C05463=1079.750,30.402,438.403,173.921,21.272,153.647
C05464=1079.745,30.152,438.419,173.920,21.270,153.647
C05465=1079.739,29.903,438.433,173.919,21.267,153.646
C05466=1079.733,29.653,438.449,173.917,21.266,153.646
C05467=1079.727,29.404,438.464,173.915,21.263,153.646
C05468=1079.722,29.154,438.479,173.914,21.260,153.646
C05469=1079.716,28.905,438.494,173.913,21.258,153.646
C05470=1079.710,28.655,438.509,173.912,21.256,153.645
C05471=1079.703,28.406,438.525,173.910,21.253,153.645
C05472=1079.698,28.157,438.540,173.908,21.251,153.645
C05473=1079.692,27.907,438.555,173.907,21.249,153.645
C05474=1079.686,27.657,438.571,173.906,21.247,153.644
C05475=1079.681,27.408,438.585,173.904,21.244,153.644
C05476=1079.675,27.158,438.601,173.902,21.242,153.644
C05477=1079.669,26.909,438.615,173.901,21.240,153.644
C05478=1079.663,26.659,438.630,173.899,21.237,153.644
C05479=1079.657,26.409,438.646,173.898,21.235,153.643
C05480=1079.651,26.160,438.660,173.897,21.233,153.643
C05481=1079.646,25.910,438.676,173.895,21.230,153.643
C05482=1079.640,25.662,438.690,173.893,21.228,153.643
C05483=1079.634,25.412,438.705,173.892,21.225,153.642
C05484=1079.629,25.163,438.721,173.891,21.223,153.642
C05485=1079.622,24.913,438.736,173.890,21.221,153.642
C05486=1079.617,24.663,438.751,173.887,21.218,153.642
C05487=1079.611,24.414,438.766,173.886,21.216,153.641
C05488=1079.604,24.164,438.781,173.885,21.214,153.641
C05489=1079.599,23.915,438.796,173.884,21.212,153.641
C05490=1079.593,23.665,438.811,173.882,21.209,153.641
C05491=1079.587,23.416,438.825,173.881,21.207,153.641
C05492=1079.581,23.167,438.841,173.879,21.205,153.640
C05493=1079.576,22.918,438.855,173.878,21.202,153.640
C05494=1079.569,22.668,438.870,173.876,21.200,153.640
C05495=1079.564,22.418,438.886,173.875,21.197,153.640
C05496=1079.558,22.169,438.901,173.873,21.195,153.640
C05497=1079.553,21.918,438.915,173.872,21.193,153.639
C05498=1079.547,21.669,438.930,173.870,21.190,153.639
C05499=1079.540,21.420,438.945,173.869,21.188,153.639
C05500=1079.535,21.171,438.960,173.868,21.186,153.639
C05501=1079.529,20.921,438.975,173.866,21.184,153.638
C05502=1079.523,20.672,438.990,173.864,21.181,153.638
C05503=1079.518,20.422,439.005,173.863,21.179,153.638
C05504=1079.512,20.172,439.019,173.862,21.177,153.638
C05505=1079.506,19.923,439.034,173.861,21.174,153.637
C05506=1079.500,19.674,439.048,173.858,21.172,153.637
C05507=1079.494,19.424,439.064,173.857,21.169,153.637
C05508=1079.488,19.175,439.079,173.856,21.167,153.637
C05509=1079.482,18.925,439.094,173.855,21.165,153.637
C05510=1079.477,18.676,439.107,173.853,21.162,153.636
C05511=1079.470,18.426,439.122,173.851,21.161,153.636
C05512=1079.465,18.177,439.138,173.850,21.158,153.636
C05513=1079.459,17.927,439.152,173.849,21.156,153.636
C05514=1079.453,17.677,439.166,173.847,21.153,153.635
C05515=1079.447,17.428,439.181,173.846,21.151,153.635
C05516=1079.442,17.179,439.196,173.844,21.149,153.635
C05517=1079.436,16.930,439.211,173.843,21.147,153.635
C05518=1079.430,16.679,439.225,173.841,21.144,153.635
C05519=1079.424,16.430,439.240,173.840,21.142,153.634
C05520=1079.418,16.181,439.255,173.839,21.139,153.634
C05521=1079.412,15.932,439.269,173.837,21.137,153.634
C05522=1079.407,15.681,439.284,173.836,21.135,153.634
C05523=1079.401,15.432,439.299,173.834,21.133,153.634
C05524=1079.395,15.154,439.315,173.833,21.130,153.633
C05525=1079.388,14.875,439.332,173.831,21.127,153.633
C05526=1079.382,14.596,439.348,173.830,21.125,153.633
C05527=1079.375,14.317,439.364,173.828,21.122,153.633
C05528=1079.369,14.068,439.378,173.826,21.120,153.632
C05529=1079.362,13.819,439.393,173.825,21.118,153.632
C05530=1079.357,13.569,439.407,173.824,21.116,153.632
C05531=1079.351,13.320,439.422,173.822,21.113,153.632
C05532=1079.345,13.070,439.436,173.820,21.111,153.631
C05533=1079.339,12.820,439.451,173.819,21.108,153.631
C05534=1079.333,12.571,439.465,173.818,21.106,153.631
C05535=1079.327,12.321,439.480,173.816,21.104,153.631
C05536=1079.321,12.072,439.494,173.815,21.102,153.631
C05537=1079.315,11.822,439.508,173.813,21.100,153.630
C05538=1079.309,11.573,439.523,173.812,21.097,153.630
C05539=1079.303,11.324,439.538,173.811,21.095,153.630
C05540=1079.297,11.074,439.552,173.809,21.092,153.630
C05541=1079.292,10.825,439.566,173.808,21.090,153.630
C05542=1079.285,10.574,439.581,173.806,21.088,153.629
C05543=1079.280,10.326,439.595,173.805,21.086,153.629
C05544=1079.274,10.075,439.609,173.803,21.083,153.629
C05545=1079.268,9.826,439.624,173.802,21.081,153.629
C05546=1079.262,9.577,439.638,173.801,21.079,153.628
C05547=1079.256,9.327,439.653,173.799,21.077,153.628
C05548=1079.250,9.077,439.667,173.797,21.074,153.628
C05549=1079.244,8.828,439.682,173.796,21.072,153.628
C05550=1079.239,8.578,439.695,173.795,21.070,153.628
C05551=1079.233,8.329,439.710,173.793,21.068,153.627
C05552=1079.227,8.079,439.724,173.792,21.066,153.627
C05553=1079.221,7.830,439.739,173.790,21.063,153.627
C05554=1079.216,7.580,439.753,173.789,21.061,153.627
C05555=1079.209,7.331,439.768,173.788,21.058,153.626
C05556=1079.204,7.081,439.782,173.786,21.056,153.626
C05557=1079.197,6.833,439.795,173.784,21.053,153.626
C05558=1079.191,6.582,439.810,173.783,21.051,153.626
C05559=1079.186,6.333,439.824,173.782,21.049,153.626
C05560=1079.180,6.084,439.838,173.781,21.047,153.625
C05561=1079.174,5.834,439.852,173.779,21.045,153.625
C05562=1079.168,5.585,439.867,173.777,21.042,153.625
C05563=1079.162,5.335,439.881,173.776,21.040,153.625
C05564=1079.156,5.085,439.895,173.775,21.038,153.625
C05565=1079.151,4.836,439.910,173.774,21.036,153.624
C05566=1079.145,4.586,439.924,173.772,21.034,153.624
C05567=1079.139,4.336,439.938,173.770,21.031,153.624
C05568=1079.133,4.087,439.952,173.769,21.029,153.624
C05569=1079.127,3.838,439.966,173.768,21.026,153.623
C05570=1079.121,3.588,439.981,173.766,21.024,153.623
C05571=1079.115,3.338,439.994,173.764,21.021,153.623
C05572=1079.110,3.089,440.008,173.763,21.019,153.623
C05573=1079.104,2.839,440.022,173.762,21.017,153.623
C05574=1079.098,2.590,440.037,173.761,21.015,153.622
C05575=1079.092,2.340,440.051,173.759,21.013,153.622
C05576=1079.086,2.091,440.064,173.757,21.010,153.622
C05577=1079.080,1.842,440.079,173.756,21.008,153.622
C05578=1079.074,1.592,440.093,173.755,21.005,153.622
C05579=1079.069,1.342,440.107,173.754,21.004,153.621
C05580=1079.063,1.092,440.121,173.752,21.002,153.621
C05581=1079.058,0.843,440.135,173.750,20.999,153.621
C05582=1079.051,0.593,440.150,173.749,20.997,153.621
C05583=1079.045,0.344,440.163,173.748,20.994,153.620
C05584=1079.040,0.094,440.177,173.747,20.992,153.620
C05585=1079.034,-0.155,440.191,173.745,20.989,153.620
C05586=1079.028,-0.405,440.206,173.743,20.987,153.620
C05587=1079.022,-0.654,440.219,173.742,20.985,153.620
C05588=1079.017,-0.931,440.234,173.741,20.983,153.619
C05589=1079.010,-1.208,440.251,173.739,20.980,153.619
C05590=1079.003,-1.484,440.265,173.738,20.977,153.619
C05591=1078.996,-1.761,440.281,173.736,20.975,153.619
C05592=1078.991,-2.011,440.295,173.734,20.972,153.618
C05593=1078.985,-2.260,440.309,173.733,20.970,153.618
C05594=1078.980,-2.510,440.323,173.732,20.968,153.618
C05595=1078.974,-2.759,440.336,173.730,20.966,153.618
C05596=1078.968,-3.009,440.350,173.729,20.963,153.618
C05597=1078.962,-3.258,440.365,173.727,20.961,153.617
C05598=1078.956,-3.508,440.379,173.726,20.959,153.617
C05599=1078.950,-3.757,440.392,173.725,20.957,153.617
C05600=1078.945,-4.007,440.406,173.723,20.954,153.617
C05601=1078.938,-4.257,440.420,173.721,20.952,153.617
C05602=1078.932,-4.506,440.434,173.720,20.950,153.616
C05603=1078.927,-4.756,440.447,173.719,20.948,153.616
C05604=1078.921,-5.005,440.461,173.718,20.946,153.616
C05605=1078.915,-5.255,440.475,173.716,20.943,153.616
C05606=1078.908,-5.505,440.488,173.714,20.941,153.616
C05607=1078.903,-5.754,440.502,173.713,20.939,153.615
C05608=1078.897,-6.004,440.516,173.712,20.937,153.615
C05609=1078.891,-6.252,440.530,173.711,20.934,153.615
C05610=1078.885,-6.503,440.544,173.708,20.932,153.615
C05611=1078.879,-6.752,440.557,173.707,20.930,153.615
C05612=1078.873,-7.002,440.571,173.706,20.928,153.614
C05613=1078.867,-7.251,440.585,173.705,20.926,153.614
C05614=1078.862,-7.500,440.598,173.703,20.924,153.614
C05615=1078.855,-7.750,440.612,173.701,20.921,153.614
C05616=1078.849,-8.000,440.626,173.700,20.919,153.614
C05617=1078.843,-8.249,440.639,173.699,20.917,153.613
C05618=1078.838,-8.499,440.653,173.698,20.914,153.613
C05619=1078.832,-8.749,440.666,173.696,20.912,153.613
C05620=1078.826,-8.998,440.679,173.695,20.910,153.613
C05621=1078.821,-9.248,440.693,173.693,20.907,153.612
C05622=1078.814,-9.497,440.707,173.692,20.905,153.612
C05623=1078.808,-9.747,440.721,173.690,20.903,153.612
C05624=1078.802,-9.997,440.734,173.689,20.901,153.612
C05625=1078.797,-10.246,440.748,173.688,20.899,153.612
C05626=1078.790,-10.495,440.761,173.686,20.896,153.612
C05627=1078.785,-10.745,440.775,173.684,20.895,153.611
C05628=1078.779,-10.994,440.788,173.683,20.892,153.611
C05629=1078.773,-11.244,440.802,173.682,20.890,153.611
C05630=1078.767,-11.493,440.815,173.681,20.888,153.611
C05631=1078.761,-11.744,440.829,173.679,20.885,153.611
C05632=1078.755,-11.993,440.842,173.677,20.883,153.610
C05633=1078.750,-12.243,440.856,173.676,20.881,153.610
C05634=1078.743,-12.492,440.869,173.675,20.879,153.610
C05635=1078.738,-12.742,440.883,173.674,20.877,153.610
C05636=1078.732,-12.991,440.897,173.672,20.874,153.610
C05637=1078.727,-13.241,440.910,173.670,20.872,153.609
C05638=1078.720,-13.490,440.923,173.669,20.870,153.609
C05639=1078.715,-13.740,440.937,173.668,20.868,153.609
C05640=1078.709,-13.989,440.950,173.666,20.866,153.609
C05641=1078.703,-14.239,440.964,173.665,20.863,153.608
C05642=1078.697,-14.488,440.977,173.663,20.861,153.608
C05643=1078.692,-14.738,440.990,173.662,20.859,153.608
C05644=1078.686,-14.988,441.004,173.661,20.856,153.608
C05645=1078.679,-15.238,441.017,173.659,20.854,153.608
C05646=1078.673,-15.487,441.031,173.658,20.852,153.608
C05647=1078.667,-15.737,441.044,173.656,20.850,153.607
C05648=1078.661,-15.986,441.057,173.655,20.848,153.607
C05649=1078.656,-16.236,441.071,173.654,20.846,153.607
C05650=1078.649,-16.485,441.084,173.652,20.844,153.607
C05651=1078.644,-16.735,441.097,173.651,20.842,153.607
C05652=1078.637,-17.010,441.111,173.649,20.839,153.606
C05653=1078.631,-17.285,441.126,173.648,20.837,153.606
C05654=1078.624,-17.560,441.141,173.646,20.835,153.606
C05655=1078.617,-17.835,441.155,173.644,20.832,153.606
C05656=1078.612,-18.085,441.168,173.643,20.830,153.606
C05657=1078.605,-18.334,441.181,173.642,20.828,153.605
C05658=1078.600,-18.584,441.195,173.640,20.826,153.605
C05659=1078.593,-18.834,441.208,173.639,20.823,153.605
C05660=1078.587,-19.083,441.221,173.637,20.821,153.605
C05661=1078.581,-19.333,441.235,173.636,20.819,153.605
C05662=1078.576,-19.583,441.248,173.634,20.817,153.605
C05663=1078.570,-19.832,441.261,173.633,20.815,153.604
C05664=1078.563,-20.081,441.274,173.632,20.812,153.604
C05665=1078.557,-20.331,441.287,173.630,20.810,153.604
C05666=1078.552,-20.581,441.301,173.629,20.808,153.604
C05667=1078.546,-20.830,441.314,173.627,20.806,153.604
C05668=1078.540,-21.080,441.327,173.626,20.804,153.603
C05669=1078.534,-21.329,441.340,173.625,20.802,153.603
C05670=1078.528,-21.579,441.353,173.624,20.800,153.603
C05671=1078.522,-21.829,441.366,173.621,20.797,153.603
C05672=1078.516,-22.079,441.379,173.620,20.795,153.603
C05673=1078.510,-22.328,441.392,173.619,20.793,153.603
C05674=1078.505,-22.577,441.406,173.618,20.791,153.602
C05675=1078.499,-22.827,441.418,173.616,20.789,153.602
C05676=1078.493,-23.076,441.431,173.615,20.787,153.602
C05677=1078.487,-23.326,441.444,173.613,20.784,153.602
C05678=1078.481,-23.575,441.457,173.612,20.782,153.602
C05679=1078.476,-23.825,441.470,173.610,20.780,153.601
C05680=1078.470,-24.074,441.484,173.609,20.778,153.601
C05681=1078.464,-24.324,441.496,173.608,20.776,153.601
C05682=1078.458,-24.574,441.509,173.607,20.774,153.601
C05683=1078.452,-24.823,441.522,173.604,20.772,153.601
C05684=1078.446,-25.073,441.536,173.603,20.770,153.601
C05685=1078.440,-25.323,441.548,173.602,20.767,153.600
C05686=1078.434,-25.572,441.562,173.601,20.765,153.600
C05687=1078.428,-25.822,441.574,173.599,20.763,153.600
C05688=1078.422,-26.072,441.587,173.598,20.761,153.600
C05689=1078.417,-26.322,441.601,173.597,20.759,153.600
C05690=1078.411,-26.571,441.613,173.594,20.757,153.599
C05691=1078.405,-26.820,441.626,173.593,20.754,153.599
C05692=1078.399,-27.070,441.639,173.592,20.752,153.599
C05693=1078.393,-27.319,441.652,173.591,20.750,153.599
C05694=1078.387,-27.569,441.665,173.589,20.748,153.599
C05695=1078.381,-27.819,441.677,173.588,20.746,153.599
C05696=1078.375,-28.068,441.690,173.586,20.744,153.598
C05697=1078.369,-28.318,441.703,173.585,20.742,153.598
C05698=1078.363,-28.567,441.716,173.583,20.740,153.598
C05699=1078.357,-28.817,441.729,173.582,20.738,153.598
C05700=1078.351,-29.067,441.741,173.581,20.736,153.598
C05701=1078.345,-29.316,441.755,173.579,20.734,153.598
C05702=1078.339,-29.566,441.767,173.578,20.732,153.597
C05703=1078.333,-29.816,441.780,173.576,20.730,153.597
C05704=1078.327,-30.065,441.793,173.575,20.728,153.597
C05705=1078.322,-30.315,441.805,173.573,20.726,153.597
C05706=1078.316,-30.564,441.818,173.572,20.723,153.597
C05707=1078.309,-30.814,441.831,173.571,20.721,153.597
C05708=1078.304,-31.064,441.843,173.570,20.719,153.596
C05709=1078.298,-31.313,441.856,173.567,20.717,153.596
C05710=1078.292,-31.563,441.869,173.566,20.715,153.596
C05711=1078.285,-31.813,441.882,173.565,20.713,153.596
C05712=1078.280,-32.063,441.894,173.564,20.711,153.596
C05713=1078.273,-32.312,441.906,173.562,20.709,153.596
C05714=1078.267,-32.561,441.919,173.561,20.707,153.595
C05715=1078.261,-32.811,441.932,173.560,20.705,153.595
C05716=1078.255,-33.085,441.946,173.557,20.702,153.595
C05717=1078.248,-33.359,441.960,173.556,20.700,153.595
C05718=1078.242,-33.634,441.973,173.555,20.698,153.595
C05719=1078.235,-33.908,441.987,173.553,20.695,153.595
C05720=1078.229,-34.158,442.000,173.552,20.693,153.594
C05721=1078.223,-34.407,442.013,173.550,20.691,153.594
C05722=1078.218,-34.656,442.025,173.549,20.690,153.594
C05723=1078.212,-34.906,442.038,173.548,20.688,153.594
C05724=1078.206,-35.156,442.050,173.546,20.686,153.594
C05725=1078.200,-35.406,442.063,173.544,20.683,153.594
C05726=1078.194,-35.655,442.076,173.543,20.681,153.593
C05727=1078.188,-35.905,442.089,173.542,20.679,153.593
C05728=1078.183,-36.154,442.101,173.540,20.677,153.593
C05729=1078.177,-36.404,442.113,173.539,20.675,153.593
C05730=1078.171,-36.654,442.126,173.538,20.673,153.593
C05731=1078.164,-36.904,442.138,173.536,20.671,153.593
C05732=1078.159,-37.153,442.150,173.534,20.669,153.593
C05733=1078.153,-37.403,442.163,173.533,20.667,153.592
C05734=1078.147,-37.652,442.176,173.532,20.665,153.592
C05735=1078.141,-37.902,442.188,173.530,20.663,153.592
C05736=1078.135,-38.152,442.201,173.529,20.661,153.592
C05737=1078.130,-38.401,442.213,173.528,20.659,153.592
C05738=1078.124,-38.651,442.226,173.526,20.657,153.592
C05739=1078.117,-38.900,442.238,173.524,20.654,153.591
C05740=1078.111,-39.150,442.250,173.523,20.652,153.591
C05741=1078.105,-39.400,442.263,173.522,20.650,153.591
C05742=1078.099,-39.649,442.274,173.520,20.649,153.591
C05743=1078.093,-39.899,442.287,173.519,20.647,153.591
C05744=1078.087,-40.149,442.299,173.517,20.645,153.591
C05745=1078.081,-40.399,442.312,173.516,20.643,153.591
C05746=1078.075,-40.647,442.324,173.515,20.641,153.590
C05747=1078.070,-40.897,442.336,173.513,20.639,153.590
C05748=1078.064,-41.147,442.349,173.511,20.637,153.590
C05749=1078.057,-41.397,442.361,173.510,20.635,153.590
C05750=1078.051,-41.647,442.373,173.509,20.633,153.590
C05751=1078.046,-41.896,442.385,173.507,20.631,153.590
C05752=1078.039,-42.145,442.397,173.506,20.629,153.590
C05753=1078.033,-42.395,442.410,173.505,20.627,153.589
C05754=1078.027,-42.645,442.422,173.503,20.625,153.589
C05755=1078.022,-42.894,442.435,173.501,20.623,153.589
C05756=1078.015,-43.144,442.447,173.500,20.621,153.589
C05757=1078.009,-43.394,442.459,173.498,20.619,153.589
C05758=1078.004,-43.644,442.472,173.497,20.617,153.589
C05759=1077.997,-43.893,442.483,173.496,20.615,153.588
C05760=1077.992,-44.142,442.496,173.494,20.614,153.588
C05761=1077.986,-44.392,442.508,173.493,20.612,153.588
C05762=1077.980,-44.641,442.520,173.492,20.610,153.588
C05763=1077.974,-44.891,442.533,173.490,20.608,153.588
C05764=1077.967,-45.141,442.545,173.488,20.605,153.588
C05765=1077.961,-45.391,442.556,173.487,20.603,153.588
C05766=1077.956,-45.640,442.569,173.485,20.602,153.588
C05767=1077.950,-45.890,442.581,173.484,20.600,153.588
C05768=1077.944,-46.140,442.593,173.483,20.598,153.587
C05769=1077.938,-46.389,442.605,173.482,20.596,153.587
C05770=1077.932,-46.639,442.617,173.480,20.594,153.587
C05771=1077.926,-46.888,442.630,173.479,20.592,153.587
C05772=1077.920,-47.138,442.642,173.478,20.590,153.587
C05773=1077.914,-47.388,442.653,173.475,20.588,153.587
C05774=1077.908,-47.638,442.666,173.474,20.586,153.587
C05775=1077.902,-47.887,442.677,173.473,20.584,153.586
C05776=1077.896,-48.136,442.690,173.471,20.582,153.586
C05777=1077.890,-48.386,442.702,173.470,20.580,153.586
C05778=1077.885,-48.636,442.713,173.469,20.578,153.586
C05779=1077.879,-48.886,442.726,173.467,20.576,153.586
C05780=1077.873,-49.160,442.739,173.465,20.574,153.586
C05781=1077.866,-49.435,442.752,173.464,20.572,153.586
C05782=1077.859,-49.709,442.766,173.462,20.570,153.585
C05783=1077.852,-49.984,442.779,173.461,20.568,153.585
C05784=1077.847,-50.234,442.791,173.459,20.566,153.585
C05785=1077.841,-50.483,442.803,173.458,20.564,153.585
C05786=1077.834,-50.733,442.815,173.456,20.562,153.585
C05787=1077.829,-50.982,442.827,173.455,20.560,153.585
C05788=1077.822,-51.232,442.838,173.454,20.558,153.585
C05789=1077.816,-51.482,442.850,173.452,20.557,153.585
C05790=1077.810,-51.732,442.862,173.451,20.555,153.584
C05791=1077.804,-51.981,442.874,173.449,20.553,153.584
C05792=1077.797,-52.231,442.885,173.448,20.551,153.584
C05793=1077.792,-52.481,442.898,173.447,20.549,153.584
C05794=1077.786,-52.730,442.909,173.444,20.547,153.584
C05795=1077.779,-52.980,442.921,173.443,20.545,153.584
C05796=1077.773,-53.230,442.933,173.442,20.543,153.584
C05797=1077.767,-53.479,442.945,173.440,20.542,153.584
C05798=1077.761,-53.729,442.956,173.439,20.540,153.584
C05799=1077.755,-53.979,442.969,173.438,20.538,153.583
C05800=1077.749,-54.227,442.980,173.436,20.537,153.583
C05801=1077.743,-54.478,442.991,173.435,20.535,153.583
C05802=1077.737,-54.728,443.004,173.433,20.533,153.583
C05803=1077.731,-54.977,443.015,173.432,20.531,153.583
C05804=1077.724,-55.227,443.027,173.431,20.529,153.583
C05805=1077.719,-55.476,443.039,173.428,20.527,153.583
C05806=1077.713,-55.726,443.050,173.427,20.525,153.583
C05807=1077.706,-55.976,443.062,173.426,20.523,153.583
C05808=1077.700,-56.225,443.073,173.424,20.522,153.583
C05809=1077.694,-56.475,443.086,173.423,20.520,153.582
C05810=1077.688,-56.724,443.097,173.421,20.518,153.582
C05811=1077.682,-56.974,443.109,173.420,20.516,153.582
C05812=1077.676,-57.224,443.121,173.418,20.515,153.582
C05813=1077.670,-57.473,443.132,173.417,20.513,153.582
C05814=1077.664,-57.723,443.144,173.416,20.511,153.582
C05815=1077.658,-57.972,443.155,173.414,20.510,153.582
C05816=1077.652,-58.222,443.167,173.413,20.508,153.582
C05817=1077.646,-58.473,443.179,173.412,20.506,153.582
C05818=1077.640,-58.721,443.190,173.409,20.504,153.582
C05819=1077.634,-58.972,443.202,173.408,20.502,153.582
C05820=1077.628,-59.221,443.214,173.407,20.500,153.581
C05821=1077.622,-59.471,443.225,173.405,20.498,153.581
C05822=1077.616,-59.720,443.236,173.404,20.497,153.581
C05823=1077.610,-59.970,443.248,173.402,20.495,153.581
C05824=1077.603,-60.220,443.260,173.401,20.493,153.581
C05825=1077.598,-60.469,443.271,173.400,20.491,153.581
C05826=1077.591,-60.719,443.283,173.398,20.490,153.581
C05827=1077.586,-60.969,443.295,173.397,20.488,153.581
C05828=1077.579,-61.218,443.307,173.395,20.486,153.581
C05829=1077.574,-61.468,443.317,173.394,20.484,153.580
C05830=1077.567,-61.718,443.329,173.392,20.483,153.580
C05831=1077.561,-61.967,443.340,173.391,20.481,153.580
C05832=1077.556,-62.217,443.352,173.389,20.479,153.580
C05833=1077.550,-62.466,443.364,173.388,20.477,153.580
C05834=1077.543,-62.716,443.375,173.386,20.475,153.580
C05835=1077.537,-62.966,443.386,173.385,20.474,153.580
C05836=1077.532,-63.216,443.398,173.383,20.472,153.580
C05837=1077.526,-63.465,443.409,173.382,20.470,153.580
C05838=1077.519,-63.715,443.421,173.381,20.468,153.580
C05839=1077.513,-63.964,443.432,173.379,20.467,153.580
C05840=1077.507,-64.215,443.443,173.378,20.465,153.579
C05841=1077.502,-64.464,443.455,173.376,20.463,153.579
C05842=1077.495,-64.714,443.467,173.375,20.461,153.579
C05843=1077.490,-64.963,443.478,173.373,20.460,153.579
C05844=1077.483,-65.239,443.490,173.371,20.457,153.579
C05845=1077.476,-65.515,443.503,173.370,20.456,153.579
C05846=1077.470,-65.791,443.516,173.368,20.454,153.579
C05847=1077.463,-66.067,443.528,173.367,20.452,153.579
C05848=1077.457,-66.317,443.539,173.366,20.451,153.579
C05849=1077.451,-66.566,443.551,173.364,20.449,153.579
C05850=1077.445,-66.816,443.562,173.362,20.447,153.579
C05851=1077.439,-67.066,443.574,173.360,20.445,153.579
C05852=1077.434,-67.316,443.585,173.359,20.443,153.578
C05853=1077.428,-67.564,443.596,173.358,20.442,153.578
C05854=1077.421,-67.815,443.608,173.356,20.440,153.578
C05855=1077.416,-68.064,443.618,173.355,20.438,153.578
C05856=1077.409,-68.314,443.630,173.354,20.436,153.578
C05857=1077.403,-68.563,443.641,173.352,20.435,153.578
C05858=1077.398,-68.813,443.653,173.351,20.433,153.578
C05859=1077.392,-69.063,443.664,173.349,20.431,153.578
C05860=1077.386,-69.313,443.675,173.348,20.430,153.578
C05861=1077.380,-69.563,443.686,173.346,20.428,153.578
C05862=1077.374,-69.812,443.698,173.345,20.427,153.578
C05863=1077.368,-70.061,443.709,173.344,20.425,153.577
C05864=1077.362,-70.311,443.720,173.342,20.423,153.577
C05865=1077.357,-70.561,443.731,173.341,20.422,153.577
C05866=1077.351,-70.811,443.742,173.339,20.420,153.577
C05867=1077.344,-71.060,443.754,173.338,20.418,153.577
C05868=1077.339,-71.310,443.765,173.337,20.416,153.577
C05869=1077.333,-71.559,443.776,173.335,20.415,153.577
C05870=1077.326,-71.809,443.787,173.333,20.413,153.577
C05871=1077.321,-72.059,443.798,173.332,20.411,153.577
C05872=1077.315,-72.308,443.809,173.330,20.409,153.577
C05873=1077.309,-72.559,443.820,173.329,20.407,153.577
C05874=1077.304,-72.808,443.832,173.327,20.406,153.577
C05875=1077.298,-73.057,443.843,173.325,20.404,153.577
C05876=1077.291,-73.307,443.854,173.324,20.402,153.576
C05877=1077.285,-73.557,443.865,173.323,20.401,153.576
C05878=1077.280,-73.806,443.876,173.321,20.400,153.576
C05879=1077.273,-74.057,443.887,173.320,20.398,153.576
C05880=1077.268,-74.306,443.898,173.318,20.396,153.576
C05881=1077.262,-74.556,443.909,173.317,20.395,153.576
C05882=1077.256,-74.806,443.920,173.315,20.393,153.576
C05883=1077.250,-75.055,443.931,173.314,20.391,153.576
C05884=1077.244,-75.305,443.943,173.313,20.390,153.576
C05885=1077.237,-75.555,443.953,173.311,20.388,153.576
C05886=1077.231,-75.804,443.964,173.310,20.387,153.576
C05887=1077.225,-76.054,443.975,173.308,20.385,153.576
C05888=1077.219,-76.304,443.986,173.307,20.383,153.576
C05889=1077.213,-76.553,443.997,173.305,20.382,153.576
C05890=1077.207,-76.804,444.008,173.304,20.380,153.576
C05891=1077.201,-77.053,444.019,173.302,20.379,153.576
C05892=1077.196,-77.303,444.030,173.301,20.377,153.576
C05893=1077.189,-77.553,444.041,173.299,20.376,153.576
C05894=1077.183,-77.802,444.051,173.298,20.374,153.575
C05895=1077.177,-78.051,444.062,173.296,20.373,153.575
C05896=1077.171,-78.301,444.073,173.295,20.371,153.575
C05897=1077.165,-78.551,444.084,173.294,20.369,153.575
C05898=1077.159,-78.801,444.095,173.292,20.368,153.575
C05899=1077.154,-79.050,444.106,173.291,20.366,153.575
C05900=1077.147,-79.300,444.117,173.289,20.365,153.575
C05901=1077.141,-79.549,444.128,173.287,20.363,153.575
C05902=1077.135,-79.799,444.138,173.286,20.361,153.575
C05903=1077.129,-80.049,444.150,173.285,20.360,153.575
C05904=1077.123,-80.299,444.161,173.283,20.358,153.575
C05905=1077.116,-80.548,444.171,173.282,20.357,153.575
C05906=1077.110,-80.798,444.182,173.280,20.356,153.575
C05907=1077.105,-81.048,444.192,173.279,20.354,153.575
C05908=1077.098,-81.325,444.205,173.277,20.353,153.575
C05909=1077.091,-81.604,444.217,173.275,20.351,153.575
C05910=1077.084,-81.882,444.228,173.273,20.349,153.575
C05911=1077.077,-82.160,444.240,173.272,20.348,153.575
C05912=1077.071,-82.410,444.251,173.270,20.346,153.575
C05913=1077.065,-82.659,444.262,173.269,20.344,153.575
C05914=1077.058,-82.909,444.273,173.267,20.343,153.575
C05915=1077.053,-83.159,444.283,173.266,20.341,153.575
C05916=1077.047,-83.409,444.294,173.264,20.340,153.575
C05917=1077.040,-83.658,444.304,173.263,20.339,153.575
C05918=1077.034,-83.908,444.315,173.261,20.337,153.575
C05919=1077.028,-84.158,444.326,173.260,20.336,153.575
C05920=1077.022,-84.407,444.336,173.258,20.334,153.575
C05921=1077.016,-84.658,444.347,173.257,20.333,153.575
C05922=1077.009,-84.907,444.357,173.255,20.331,153.574
C05923=1077.004,-85.156,444.368,173.254,20.330,153.574
C05924=1076.998,-85.406,444.379,173.252,20.328,153.574
C05925=1076.991,-85.656,444.389,173.251,20.327,153.574
C05926=1076.985,-85.906,444.400,173.249,20.326,153.575
C05927=1076.980,-86.155,444.411,173.248,20.324,153.575
C05928=1076.973,-86.404,444.421,173.246,20.323,153.574
C05929=1076.967,-86.655,444.431,173.245,20.322,153.574
C05930=1076.961,-86.904,444.442,173.243,20.320,153.574
C05931=1076.955,-87.154,444.453,173.241,20.319,153.574
C05932=1076.949,-87.403,444.463,173.240,20.317,153.574
C05933=1076.943,-87.653,444.473,173.238,20.316,153.574
C05934=1076.937,-87.903,444.484,173.237,20.314,153.574
C05935=1076.931,-88.153,444.495,173.235,20.313,153.574
C05936=1076.925,-88.403,444.505,173.234,20.311,153.574
C05937=1076.919,-88.652,444.516,173.232,20.310,153.574
C05938=1076.912,-88.902,444.526,173.231,20.308,153.574
C05939=1076.907,-89.152,444.536,173.229,20.307,153.574
C05940=1076.901,-89.402,444.547,173.228,20.306,153.574
C05941=1076.894,-89.651,444.558,173.226,20.304,153.574
C05942=1076.889,-89.901,444.568,173.225,20.303,153.574
C05943=1076.882,-90.150,444.578,173.223,20.302,153.574
C05944=1076.876,-90.400,444.589,173.222,20.300,153.574
C05945=1076.870,-90.650,444.599,173.220,20.299,153.574
C05946=1076.864,-90.900,444.610,173.219,20.297,153.574
C05947=1076.858,-91.149,444.621,173.217,20.296,153.574
C05948=1076.852,-91.399,444.630,173.216,20.294,153.574
C05949=1076.846,-91.648,444.641,173.214,20.293,153.574
C05950=1076.840,-91.899,444.651,173.213,20.291,153.574
C05951=1076.834,-92.148,444.662,173.212,20.291,153.574
C05952=1076.827,-92.398,444.672,173.210,20.290,153.574
C05953=1076.822,-92.648,444.682,173.209,20.288,153.574
C05954=1076.816,-92.897,444.693,173.207,20.287,153.574
C05955=1076.810,-93.147,444.703,173.206,20.285,153.574
C05956=1076.804,-93.396,444.714,173.204,20.284,153.574
C05957=1076.798,-93.646,444.723,173.202,20.283,153.574
C05958=1076.792,-93.896,444.734,173.201,20.281,153.574
C05959=1076.786,-94.146,444.744,173.199,20.280,153.574
C05960=1076.780,-94.396,444.755,173.198,20.278,153.574
C05961=1076.774,-94.645,444.764,173.196,20.277,153.574
C05962=1076.768,-94.895,444.775,173.195,20.276,153.574
C05963=1076.762,-95.145,444.785,173.193,20.275,153.574
C05964=1076.756,-95.394,444.796,173.192,20.273,153.574
C05965=1076.750,-95.644,444.805,173.190,20.272,153.574
C05966=1076.744,-95.894,444.816,173.189,20.270,153.574
C05967=1076.738,-96.143,444.826,173.187,20.269,153.574
C05968=1076.732,-96.394,444.837,173.185,20.268,153.574
C05969=1076.726,-96.643,444.847,173.184,20.266,153.574
C05970=1076.720,-96.893,444.857,173.182,20.265,153.574
C05971=1076.714,-97.143,444.867,173.181,20.263,153.574
C05972=1076.707,-97.423,444.879,173.179,20.262,153.574
C05973=1076.701,-97.703,444.890,173.178,20.261,153.574
C05974=1076.694,-97.983,444.901,173.176,20.260,153.574
C05975=1076.686,-98.263,444.913,173.175,20.258,153.574
C05976=1076.681,-98.514,444.923,173.173,20.257,153.574
C05977=1076.675,-98.763,444.933,173.171,20.256,153.574
C05978=1076.668,-99.013,444.943,173.170,20.254,153.574
C05979=1076.663,-99.263,444.953,173.168,20.253,153.574
C05980=1076.656,-99.513,444.964,173.167,20.252,153.574
C05981=1076.650,-99.762,444.973,173.165,20.251,153.574
C05982=1076.644,-100.012,444.983,173.163,20.250,153.574
C05983=1076.638,-100.262,444.994,173.162,20.248,153.574
C05984=1076.631,-100.511,445.003,173.160,20.247,153.574
C05985=1076.626,-100.761,445.014,173.159,20.246,153.575
C05986=1076.620,-101.011,445.024,173.157,20.244,153.575
C05987=1076.613,-101.261,445.033,173.155,20.243,153.575
C05988=1076.608,-101.510,445.044,173.155,20.242,153.575
C05989=1076.601,-101.760,445.054,173.153,20.241,153.575
C05990=1076.595,-102.010,445.063,173.151,20.240,153.575
C05991=1076.589,-102.259,445.074,173.150,20.239,153.575
C05992=1076.583,-102.509,445.084,173.148,20.238,153.575
C05993=1076.577,-102.759,445.093,173.147,20.236,153.575
C05994=1076.571,-103.008,445.103,173.145,20.235,153.575
C05995=1076.565,-103.259,445.114,173.143,20.234,153.575
C05996=1076.559,-103.508,445.124,173.142,20.232,153.575
C05997=1076.552,-103.758,445.133,173.140,20.231,153.575
C05998=1076.546,-104.007,445.144,173.139,20.230,153.575
C05999=1076.540,-104.258,445.154,173.137,20.229,153.575
C06000=1076.534,-104.507,445.163,173.135,20.228,153.575
C06001=1076.528,-104.757,445.173,173.135,20.227,153.575
C06002=1076.522,-105.006,445.183,173.133,20.226,153.575
C06003=1076.516,-105.256,445.193,173.131,20.225,153.575
C06004=1076.510,-105.506,445.203,173.130,20.223,153.575
C06005=1076.504,-105.756,445.212,173.128,20.222,153.575
C06006=1076.497,-106.005,445.223,173.127,20.221,153.575
C06007=1076.491,-106.255,445.232,173.125,20.220,153.575
C06008=1076.486,-106.505,445.242,173.123,20.219,153.575
C06009=1076.480,-106.755,445.252,173.122,20.218,153.575
C06010=1076.473,-107.005,445.262,173.120,20.216,153.575
C06011=1076.467,-107.254,445.272,173.118,20.215,153.576
C06012=1076.461,-107.504,445.281,173.118,20.214,153.575
C06013=1076.455,-107.754,445.292,173.116,20.213,153.576
C06014=1076.449,-108.004,445.301,173.114,20.212,153.576
C06015=1076.443,-108.253,445.311,173.113,20.211,153.576
C06016=1076.436,-108.503,445.321,173.111,20.210,153.576
C06017=1076.430,-108.752,445.331,173.110,20.209,153.576
C06018=1076.424,-109.002,445.340,173.108,20.208,153.576
C06019=1076.418,-109.252,445.350,173.106,20.207,153.576
C06020=1076.412,-109.502,445.359,173.105,20.205,153.576
C06021=1076.406,-109.752,445.369,173.103,20.204,153.576
C06022=1076.400,-110.002,445.379,173.102,20.204,153.576
C06023=1076.394,-110.251,445.389,173.100,20.202,153.576
C06024=1076.388,-110.500,445.399,173.099,20.201,153.576
C06025=1076.382,-110.750,445.408,173.097,20.201,153.576
C06026=1076.376,-111.000,445.418,173.095,20.199,153.576
C06027=1076.370,-111.249,445.427,173.094,20.198,153.577
C06028=1076.363,-111.499,445.437,173.092,20.197,153.577
C06029=1076.357,-111.749,445.446,173.091,20.196,153.577
C06030=1076.351,-111.999,445.456,173.089,20.195,153.577
C06031=1076.345,-112.249,445.465,173.088,20.194,153.577
C06032=1076.339,-112.498,445.475,173.086,20.193,153.577
C06033=1076.333,-112.748,445.485,173.085,20.192,153.577
C06034=1076.326,-112.998,445.494,173.083,20.191,153.577
C06035=1076.320,-113.248,445.504,173.081,20.190,153.577
C06036=1076.314,-113.525,445.515,173.080,20.189,153.577
C06037=1076.307,-113.803,445.525,173.078,20.188,153.577
C06038=1076.300,-114.081,445.536,173.076,20.186,153.577
C06039=1076.293,-114.358,445.546,173.075,20.185,153.577
C06040=1076.287,-114.608,445.556,173.073,20.185,153.577
C06041=1076.281,-114.858,445.565,173.071,20.184,153.578
C06042=1076.275,-115.107,445.575,173.070,20.182,153.578
C06043=1076.269,-115.357,445.585,173.068,20.181,153.578
C06044=1076.263,-115.607,445.594,173.066,20.180,153.578
C06045=1076.256,-115.857,445.604,173.065,20.180,153.578
C06046=1076.250,-116.107,445.613,173.064,20.179,153.578
C06047=1076.244,-116.356,445.623,173.062,20.177,153.578
C06048=1076.238,-116.606,445.632,173.060,20.177,153.578
C06049=1076.232,-116.855,445.642,173.059,20.176,153.578
C06050=1076.226,-117.105,445.651,173.057,20.175,153.578
C06051=1076.220,-117.355,445.661,173.055,20.174,153.578
C06052=1076.214,-117.605,445.670,173.054,20.173,153.579
C06053=1076.208,-117.855,445.680,173.053,20.172,153.578
C06054=1076.201,-118.104,445.689,173.051,20.171,153.579
C06055=1076.195,-118.354,445.699,173.049,20.170,153.579
C06056=1076.189,-118.605,445.708,173.048,20.169,153.579
C06057=1076.183,-118.853,445.716,173.046,20.168,153.579
C06058=1076.177,-119.103,445.726,173.044,20.167,153.579
C06059=1076.171,-119.353,445.736,173.042,20.166,153.579
C06060=1076.165,-119.603,445.745,173.042,20.166,153.579
C06061=1076.158,-119.853,445.755,173.040,20.164,153.579
C06062=1076.152,-120.102,445.764,173.038,20.164,153.579
C06063=1076.146,-120.352,445.774,173.037,20.163,153.579
C06064=1076.141,-120.602,445.782,173.035,20.162,153.580
C06065=1076.134,-120.851,445.791,173.033,20.161,153.580
C06066=1076.128,-121.101,445.801,173.032,20.160,153.580
C06067=1076.122,-121.351,445.810,173.031,20.159,153.580
C06068=1076.115,-121.601,445.820,173.029,20.159,153.580
C06069=1076.109,-121.851,445.830,173.027,20.158,153.580
C06070=1076.103,-122.101,445.838,173.025,20.157,153.580
C06071=1076.098,-122.350,445.848,173.024,20.156,153.580
C06072=1076.091,-122.600,445.857,173.022,20.155,153.580
C06073=1076.085,-122.849,445.866,173.021,20.154,153.581
C06074=1076.078,-123.099,445.876,173.019,20.153,153.581
C06075=1076.073,-123.350,445.885,173.018,20.153,153.581
C06076=1076.067,-123.599,445.894,173.016,20.152,153.581
C06077=1076.061,-123.848,445.903,173.014,20.151,153.581
C06078=1076.054,-124.098,445.912,173.012,20.150,153.581
C06079=1076.048,-124.348,445.921,173.012,20.149,153.581
C06080=1076.042,-124.598,445.931,173.010,20.148,153.581
C06081=1076.036,-124.848,445.940,173.008,20.148,153.581
C06082=1076.029,-125.097,445.949,173.006,20.147,153.582
C06083=1076.024,-125.347,445.958,173.005,20.146,153.582
C06084=1076.017,-125.597,445.967,173.003,20.145,153.582
C06085=1076.011,-125.847,445.977,173.002,20.144,153.582
C06086=1076.005,-126.097,445.985,173.000,20.143,153.582
C06087=1075.999,-126.346,445.994,172.999,20.142,153.582
C06088=1075.993,-126.596,446.004,172.997,20.142,153.582
C06089=1075.987,-126.846,446.013,172.995,20.141,153.582
C06090=1075.980,-127.096,446.022,172.994,20.140,153.582
C06091=1075.974,-127.345,446.031,172.992,20.140,153.583
C06092=1075.968,-127.596,446.040,172.990,20.139,153.583
C06093=1075.962,-127.846,446.050,172.989,20.138,153.583
C06094=1075.956,-128.096,446.059,172.987,20.137,153.583
C06095=1075.954,-128.347,446.069,172.986,20.135,153.583
C06096=1075.953,-128.601,446.080,172.985,20.132,153.582
C06097=1075.956,-128.855,446.093,172.984,20.129,153.582
C06098=1075.961,-129.106,446.107,172.984,20.124,153.581
C06099=1075.968,-129.358,446.121,172.984,20.119,153.580
C06100=1075.573,-129.380,445.969,172.939,20.248,153.611
C06101=1075.565,-129.129,445.955,172.939,20.253,153.612
C06102=1075.561,-128.876,445.941,172.940,20.257,153.613
C06103=1075.558,-128.623,445.929,172.940,20.261,153.614
C06104=1075.559,-128.368,445.917,172.941,20.264,153.614
C06105=1075.561,-128.119,445.906,172.942,20.266,153.614
C06106=1075.566,-127.868,445.896,172.944,20.267,153.614
C06107=1075.572,-127.618,445.887,172.946,20.268,153.614
C06108=1075.578,-127.367,445.878,172.947,20.268,153.614
C06109=1075.584,-127.118,445.870,172.948,20.269,153.614
C06110=1075.591,-126.868,445.860,172.950,20.270,153.614
C06111=1075.596,-126.618,445.851,172.952,20.271,153.613
C06112=1075.603,-126.368,445.842,172.954,20.272,153.613
C06113=1075.609,-126.119,445.833,172.956,20.272,153.613
C06114=1075.615,-125.869,445.824,172.956,20.273,153.613
C06115=1075.621,-125.619,445.815,172.958,20.274,153.613
C06116=1075.628,-125.369,445.806,172.960,20.275,153.613
C06117=1075.634,-125.119,445.796,172.962,20.276,153.613
C06118=1075.640,-124.869,445.787,172.963,20.277,153.613
C06119=1075.646,-124.620,445.779,172.965,20.277,153.612
C06120=1075.652,-124.370,445.769,172.966,20.278,153.612
C06121=1075.659,-124.121,445.759,172.968,20.279,153.612
C06122=1075.664,-123.870,445.751,172.969,20.280,153.612
C06123=1075.671,-123.620,445.741,172.971,20.281,153.612
C06124=1075.676,-123.371,445.732,172.973,20.282,153.612
C06125=1075.683,-123.122,445.723,172.975,20.282,153.612
C06126=1075.689,-122.871,445.714,172.975,20.283,153.612
C06127=1075.695,-122.622,445.704,172.977,20.284,153.612
C06128=1075.701,-122.372,445.695,172.979,20.285,153.611
C06129=1075.707,-122.122,445.685,172.981,20.286,153.611
C06130=1075.713,-121.873,445.676,172.982,20.287,153.611
C06131=1075.720,-121.623,445.668,172.984,20.287,153.611
C06132=1075.726,-121.373,445.658,172.985,20.288,153.611
C06133=1075.732,-121.123,445.649,172.987,20.289,153.611
C06134=1075.738,-120.873,445.639,172.988,20.290,153.611
C06135=1075.744,-120.624,445.630,172.990,20.291,153.611
C06136=1075.750,-120.375,445.620,172.992,20.292,153.611
C06137=1075.756,-120.125,445.611,172.993,20.293,153.611
C06138=1075.763,-119.875,445.603,172.995,20.294,153.610
C06139=1075.769,-119.625,445.593,172.996,20.294,153.610
C06140=1075.775,-119.375,445.583,172.998,20.295,153.610
C06141=1075.781,-119.125,445.574,173.000,20.296,153.610
C06142=1075.787,-118.875,445.564,173.001,20.298,153.610
C06143=1075.794,-118.626,445.555,173.003,20.299,153.610
C06144=1075.799,-118.377,445.546,173.005,20.299,153.610
C06145=1075.805,-118.127,445.536,173.006,20.300,153.610
C06146=1075.811,-117.877,445.526,173.007,20.301,153.610
C06147=1075.817,-117.627,445.518,173.009,20.302,153.610
C06148=1075.824,-117.377,445.508,173.010,20.303,153.610
C06149=1075.830,-117.127,445.499,173.012,20.304,153.610
C06150=1075.837,-116.877,445.489,173.014,20.305,153.609
C06151=1075.843,-116.628,445.480,173.016,20.306,153.609
C06152=1075.849,-116.378,445.470,173.017,20.307,153.609
C06153=1075.855,-116.129,445.461,173.019,20.308,153.609
C06154=1075.861,-115.879,445.452,173.020,20.309,153.609
C06155=1075.867,-115.629,445.442,173.021,20.310,153.609
C06156=1075.873,-115.379,445.432,173.023,20.311,153.609
C06157=1075.879,-115.130,445.423,173.025,20.311,153.609
C06158=1075.885,-114.880,445.413,173.026,20.313,153.609
C06159=1075.892,-114.630,445.404,173.028,20.314,153.609
C06160=1075.898,-114.380,445.394,173.030,20.315,153.609
C06161=1075.905,-114.102,445.384,173.031,20.316,153.609
C06162=1075.911,-113.825,445.373,173.033,20.317,153.609
C06163=1075.918,-113.547,445.362,173.035,20.318,153.608
C06164=1075.925,-113.269,445.351,173.036,20.319,153.608
C06165=1075.931,-113.019,445.342,173.038,20.320,153.608
C06166=1075.938,-112.770,445.332,173.040,20.321,153.608
C06167=1075.943,-112.520,445.323,173.042,20.322,153.608
C06168=1075.949,-112.271,445.313,173.043,20.324,153.608
C06169=1075.955,-112.021,445.303,173.044,20.324,153.608
C06170=1075.961,-111.771,445.294,173.046,20.325,153.608
C06171=1075.967,-111.521,445.284,173.047,20.326,153.608
C06172=1075.973,-111.271,445.274,173.049,20.327,153.608
C06173=1075.979,-111.021,445.265,173.051,20.329,153.608
C06174=1075.986,-110.772,445.255,173.052,20.330,153.608
C06175=1075.992,-110.522,445.246,173.054,20.331,153.608
C06176=1075.998,-110.272,445.236,173.055,20.332,153.608
C06177=1076.004,-110.023,445.226,173.057,20.333,153.607
C06178=1076.011,-109.773,445.216,173.058,20.333,153.607
C06179=1076.017,-109.523,445.207,173.060,20.335,153.607
C06180=1076.023,-109.273,445.197,173.061,20.336,153.607
C06181=1076.028,-109.023,445.187,173.063,20.337,153.607
C06182=1076.035,-108.773,445.177,173.065,20.338,153.607
C06183=1076.041,-108.524,445.168,173.066,20.339,153.607
C06184=1076.047,-108.274,445.158,173.068,20.341,153.607
C06185=1076.053,-108.025,445.148,173.070,20.341,153.607
C06186=1076.060,-107.775,445.138,173.071,20.343,153.607
C06187=1076.066,-107.525,445.129,173.073,20.344,153.607
C06188=1076.072,-107.275,445.119,173.074,20.345,153.607
C06189=1076.077,-107.025,445.109,173.075,20.346,153.607
C06190=1076.084,-106.776,445.099,173.077,20.347,153.607
C06191=1076.090,-106.526,445.089,173.078,20.348,153.607
C06192=1076.096,-106.276,445.080,173.080,20.350,153.607
C06193=1076.102,-106.027,445.070,173.082,20.350,153.607
C06194=1076.108,-105.777,445.059,173.083,20.352,153.607
C06195=1076.114,-105.527,445.050,173.085,20.353,153.607
C06196=1076.120,-105.278,445.040,173.086,20.354,153.607
C06197=1076.127,-105.028,445.031,173.088,20.355,153.606
C06198=1076.132,-104.778,445.020,173.090,20.357,153.607
C06199=1076.138,-104.528,445.010,173.091,20.358,153.606
C06200=1076.145,-104.279,445.001,173.092,20.359,153.606
C06201=1076.151,-104.029,444.991,173.094,20.359,153.606
C06202=1076.157,-103.779,444.980,173.095,20.361,153.606
C06203=1076.163,-103.530,444.971,173.097,20.362,153.606
C06204=1076.169,-103.280,444.961,173.099,20.363,153.606
C06205=1076.175,-103.030,444.951,173.100,20.365,153.606
C06206=1076.181,-102.780,444.941,173.102,20.366,153.606
C06207=1076.187,-102.531,444.931,173.103,20.367,153.606
C06208=1076.193,-102.281,444.921,173.105,20.368,153.606
C06209=1076.199,-102.031,444.911,173.107,20.369,153.606
C06210=1076.205,-101.782,444.901,173.108,20.371,153.606
C06211=1076.211,-101.532,444.891,173.110,20.372,153.606
C06212=1076.218,-101.283,444.881,173.111,20.373,153.606
C06213=1076.224,-101.032,444.871,173.113,20.374,153.606
C06214=1076.230,-100.782,444.861,173.114,20.375,153.606
C06215=1076.236,-100.533,444.851,173.115,20.377,153.606
C06216=1076.242,-100.283,444.841,173.117,20.378,153.606
C06217=1076.248,-100.034,444.830,173.119,20.379,153.606
C06218=1076.254,-99.784,444.821,173.120,20.380,153.606
C06219=1076.260,-99.534,444.811,173.122,20.381,153.606
C06220=1076.266,-99.284,444.800,173.123,20.383,153.606
C06221=1076.273,-99.035,444.791,173.125,20.384,153.606
C06222=1076.278,-98.785,444.780,173.127,20.385,153.606
C06223=1076.284,-98.535,444.770,173.128,20.387,153.606
C06224=1076.291,-98.285,444.760,173.130,20.388,153.606
C06225=1076.298,-98.006,444.749,173.131,20.389,153.606
C06226=1076.304,-97.725,444.737,173.133,20.390,153.606
C06227=1076.311,-97.444,444.726,173.134,20.392,153.606
C06228=1076.318,-97.163,444.715,173.137,20.394,153.606
C06229=1076.324,-96.914,444.704,173.138,20.395,153.606
C06230=1076.330,-96.664,444.695,173.139,20.396,153.606
C06231=1076.336,-96.415,444.684,173.141,20.397,153.606
C06232=1076.343,-96.164,444.674,173.142,20.399,153.606
C06233=1076.348,-95.915,444.663,173.144,20.400,153.606
C06234=1076.354,-95.665,444.653,173.145,20.402,153.606
C06235=1076.360,-95.415,444.643,173.147,20.402,153.606
C06236=1076.366,-95.165,444.632,173.148,20.404,153.606
C06237=1076.372,-94.916,444.622,173.150,20.405,153.606
C06238=1076.378,-94.666,444.612,173.151,20.407,153.606
C06239=1076.384,-94.417,444.602,173.153,20.408,153.606
C06240=1076.390,-94.167,444.592,173.155,20.410,153.606
C06241=1076.396,-93.917,444.581,173.156,20.411,153.606
C06242=1076.402,-93.667,444.571,173.158,20.412,153.606
C06243=1076.409,-93.418,444.560,173.159,20.414,153.606
C06244=1076.414,-93.168,444.550,173.161,20.415,153.606
C06245=1076.421,-92.918,444.540,173.162,20.416,153.606
C06246=1076.426,-92.669,444.529,173.164,20.418,153.606
C06247=1076.432,-92.419,444.519,173.165,20.419,153.606
C06248=1076.438,-92.169,444.509,173.167,20.421,153.606
C06249=1076.444,-91.919,444.499,173.169,20.422,153.606
C06250=1076.451,-91.669,444.488,173.170,20.423,153.606
C06251=1076.456,-91.420,444.477,173.172,20.425,153.606
C06252=1076.463,-91.170,444.467,173.173,20.426,153.606
C06253=1076.468,-90.921,444.457,173.175,20.428,153.606
C06254=1076.475,-90.672,444.446,173.176,20.429,153.606
C06255=1076.480,-90.421,444.436,173.178,20.430,153.606
C06256=1076.487,-90.171,444.425,173.179,20.432,153.606
C06257=1076.493,-89.921,444.415,173.181,20.433,153.606
C06258=1076.498,-89.672,444.404,173.181,20.434,153.606
C06259=1076.505,-89.423,444.394,173.183,20.436,153.606
C06260=1076.510,-89.173,444.384,173.185,20.437,153.606
C06261=1076.517,-88.922,444.373,173.186,20.438,153.606
C06262=1076.523,-88.673,444.362,173.188,20.440,153.606
C06263=1076.529,-88.423,444.352,173.189,20.441,153.606
C06264=1076.535,-88.174,444.342,173.191,20.443,153.606
C06265=1076.541,-87.924,444.331,173.192,20.444,153.606
C06266=1076.547,-87.674,444.320,173.194,20.445,153.606
C06267=1076.553,-87.424,444.310,173.195,20.447,153.606
C06268=1076.559,-87.175,444.299,173.197,20.448,153.606
C06269=1076.566,-86.926,444.289,173.198,20.450,153.606
C06270=1076.571,-86.676,444.279,173.200,20.451,153.606
C06271=1076.577,-86.426,444.268,173.201,20.453,153.606
C06272=1076.584,-86.176,444.257,173.203,20.454,153.606
C06273=1076.590,-85.927,444.247,173.204,20.456,153.606
C06274=1076.595,-85.677,444.236,173.206,20.457,153.606
C06275=1076.602,-85.427,444.226,173.207,20.458,153.606
C06276=1076.608,-85.177,444.215,173.209,20.460,153.606
C06277=1076.614,-84.928,444.205,173.210,20.461,153.606
C06278=1076.621,-84.678,444.193,173.212,20.463,153.606
C06279=1076.626,-84.428,444.183,173.213,20.464,153.606
C06280=1076.633,-84.179,444.173,173.215,20.466,153.606
C06281=1076.638,-83.929,444.162,173.216,20.467,153.606
C06282=1076.645,-83.679,444.151,173.218,20.469,153.606
C06283=1076.651,-83.430,444.141,173.220,20.470,153.606
C06284=1076.657,-83.180,444.130,173.221,20.472,153.606
C06285=1076.663,-82.930,444.119,173.223,20.473,153.606
C06286=1076.669,-82.680,444.109,173.224,20.474,153.606
C06287=1076.675,-82.431,444.098,173.226,20.476,153.606
C06288=1076.681,-82.181,444.087,173.227,20.477,153.606
C06289=1076.688,-81.903,444.075,173.228,20.479,153.607
C06290=1076.695,-81.625,444.064,173.231,20.481,153.607
C06291=1076.702,-81.346,444.052,173.232,20.483,153.607
C06292=1076.709,-81.069,444.040,173.234,20.484,153.607
C06293=1076.715,-80.818,444.029,173.235,20.486,153.607
C06294=1076.721,-80.569,444.018,173.237,20.487,153.607
C06295=1076.728,-80.319,444.007,173.238,20.488,153.607
C06296=1076.733,-80.069,443.996,173.240,20.490,153.607
C06297=1076.739,-79.820,443.985,173.241,20.492,153.607
C06298=1076.745,-79.570,443.974,173.243,20.493,153.607
C06299=1076.752,-79.321,443.964,173.244,20.495,153.607
C06300=1076.758,-79.071,443.953,173.246,20.496,153.607
C06301=1076.763,-78.821,443.943,173.247,20.498,153.607
C06302=1076.770,-78.571,443.932,173.249,20.500,153.607
C06303=1076.775,-78.321,443.921,173.250,20.501,153.607
C06304=1076.781,-78.072,443.910,173.252,20.503,153.607
C06305=1076.787,-77.822,443.899,173.253,20.504,153.607
C06306=1076.793,-77.572,443.888,173.254,20.506,153.607
C06307=1076.800,-77.323,443.877,173.256,20.508,153.607
C06308=1076.806,-77.073,443.866,173.257,20.509,153.607
C06309=1076.812,-76.823,443.855,173.259,20.510,153.607
C06310=1076.817,-76.574,443.844,173.261,20.512,153.607
C06311=1076.824,-76.324,443.833,173.262,20.514,153.608
C06312=1076.829,-76.074,443.822,173.263,20.515,153.608
C06313=1076.835,-75.825,443.811,173.265,20.517,153.608
C06314=1076.842,-75.574,443.800,173.266,20.518,153.608
C06315=1076.848,-75.326,443.789,173.268,20.520,153.608
C06316=1076.854,-75.076,443.778,173.270,20.522,153.608
C06317=1076.860,-74.826,443.767,173.272,20.524,153.608
C06318=1076.866,-74.577,443.756,173.273,20.525,153.608
C06319=1076.872,-74.327,443.745,173.274,20.527,153.608
C06320=1076.878,-74.077,443.734,173.276,20.528,153.608
C06321=1076.884,-73.828,443.723,173.277,20.530,153.608
C06322=1076.890,-73.577,443.712,173.279,20.532,153.608
C06323=1076.896,-73.328,443.701,173.280,20.533,153.608
C06324=1076.902,-73.078,443.690,173.282,20.535,153.608
C06325=1076.907,-72.829,443.679,173.283,20.537,153.608
C06326=1076.913,-72.578,443.667,173.285,20.538,153.608
C06327=1076.919,-72.330,443.656,173.286,20.540,153.609
C06328=1076.925,-72.080,443.645,173.287,20.542,153.609
C06329=1076.931,-71.830,443.634,173.289,20.544,153.609
C06330=1076.937,-71.580,443.623,173.290,20.545,153.609
C06331=1076.943,-71.330,443.612,173.292,20.547,153.609
C06332=1076.949,-71.081,443.601,173.293,20.549,153.609
C06333=1076.955,-70.831,443.590,173.295,20.550,153.609
C06334=1076.961,-70.581,443.577,173.296,20.552,153.609
C06335=1076.966,-70.332,443.566,173.297,20.553,153.609
C06336=1076.972,-70.082,443.556,173.299,20.555,153.609
C06337=1076.979,-69.832,443.544,173.300,20.557,153.609
C06338=1076.984,-69.583,443.533,173.302,20.559,153.610
C06339=1076.990,-69.334,443.522,173.303,20.560,153.610
C06340=1076.997,-69.084,443.511,173.305,20.562,153.610
C06341=1077.002,-68.834,443.499,173.307,20.564,153.610
C06342=1077.008,-68.584,443.488,173.308,20.566,153.610
C06343=1077.014,-68.335,443.476,173.310,20.568,153.610
C06344=1077.020,-68.085,443.465,173.311,20.569,153.610
C06345=1077.026,-67.835,443.454,173.312,20.571,153.610
C06346=1077.032,-67.586,443.443,173.314,20.572,153.610
C06347=1077.039,-67.336,443.431,173.315,20.574,153.610
C06348=1077.044,-67.086,443.420,173.317,20.576,153.610
C06349=1077.050,-66.836,443.409,173.318,20.578,153.610
C06350=1077.056,-66.586,443.398,173.320,20.579,153.610
C06351=1077.062,-66.338,443.386,173.321,20.581,153.611
C06352=1077.068,-66.087,443.375,173.322,20.583,153.611
C06353=1077.074,-65.811,443.362,173.324,20.585,153.611
C06354=1077.081,-65.535,443.349,173.326,20.587,153.611
C06355=1077.087,-65.259,443.337,173.327,20.589,153.611
C06356=1077.094,-64.983,443.325,173.329,20.591,153.611
C06357=1077.100,-64.734,443.313,173.330,20.592,153.611
C06358=1077.106,-64.484,443.301,173.331,20.594,153.611
C06359=1077.112,-64.234,443.291,173.333,20.596,153.611
C06360=1077.118,-63.985,443.279,173.334,20.598,153.611
C06361=1077.124,-63.735,443.268,173.336,20.599,153.611
C06362=1077.130,-63.485,443.256,173.338,20.601,153.612
C06363=1077.136,-63.236,443.244,173.339,20.603,153.612
C06364=1077.142,-62.986,443.233,173.341,20.605,153.612
C06365=1077.148,-62.737,443.221,173.342,20.607,153.612
C06366=1077.154,-62.487,443.210,173.344,20.608,153.612
C06367=1077.159,-62.237,443.199,173.345,20.610,153.612
C06368=1077.166,-61.987,443.187,173.346,20.612,153.612
C06369=1077.172,-61.738,443.176,173.348,20.614,153.612
C06370=1077.178,-61.488,443.164,173.349,20.615,153.612
C06371=1077.183,-61.238,443.152,173.351,20.617,153.612
C06372=1077.190,-60.989,443.140,173.352,20.619,153.613
C06373=1077.196,-60.739,443.130,173.353,20.621,153.613
C06374=1077.202,-60.489,443.118,173.355,20.623,153.613
C06375=1077.208,-60.239,443.106,173.356,20.624,153.613
C06376=1077.214,-59.990,443.095,173.358,20.626,153.613
C06377=1077.220,-59.740,443.083,173.360,20.628,153.613
C06378=1077.226,-59.491,443.072,173.361,20.630,153.613
C06379=1077.232,-59.241,443.060,173.363,20.632,153.613
C06380=1077.238,-58.991,443.049,173.364,20.633,153.613
C06381=1077.244,-58.742,443.037,173.365,20.635,153.614
C06382=1077.250,-58.492,443.026,173.367,20.637,153.614
C06383=1077.256,-58.242,443.013,173.368,20.639,153.614
C06384=1077.262,-57.992,443.002,173.370,20.641,153.614
C06385=1077.268,-57.743,442.990,173.371,20.642,153.614
C06386=1077.275,-57.494,442.978,173.372,20.644,153.614
C06387=1077.280,-57.244,442.967,173.374,20.646,153.614
C06388=1077.287,-56.994,442.955,173.375,20.648,153.614
C06389=1077.293,-56.744,442.944,173.377,20.650,153.614
C06390=1077.298,-56.495,442.932,173.379,20.651,153.614
C06391=1077.305,-56.245,442.920,173.380,20.653,153.615
C06392=1077.311,-55.996,442.909,173.382,20.655,153.615
C06393=1077.317,-55.746,442.897,173.383,20.657,153.615
C06394=1077.323,-55.496,442.885,173.384,20.659,153.615
C06395=1077.329,-55.247,442.873,173.386,20.660,153.615
C06396=1077.335,-54.997,442.862,173.387,20.662,153.615
C06397=1077.341,-54.747,442.850,173.388,20.664,153.615
C06398=1077.347,-54.498,442.838,173.390,20.666,153.615
C06399=1077.354,-54.248,442.827,173.391,20.668,153.615
C06400=1077.360,-53.998,442.814,173.393,20.670,153.616
C06401=1077.366,-53.749,442.803,173.395,20.672,153.616
C06402=1077.372,-53.499,442.791,173.396,20.674,153.616
C06403=1077.378,-53.249,442.779,173.398,20.676,153.616
C06404=1077.384,-53.000,442.767,173.399,20.677,153.616
C06405=1077.390,-52.750,442.756,173.400,20.679,153.616
C06406=1077.396,-52.500,442.743,173.402,20.681,153.616
C06407=1077.402,-52.251,442.732,173.403,20.682,153.616
C06408=1077.409,-52.001,442.721,173.405,20.684,153.616
C06409=1077.415,-51.751,442.708,173.406,20.686,153.617
C06410=1077.421,-51.502,442.696,173.407,20.688,153.617
C06411=1077.427,-51.253,442.684,173.409,20.690,153.617
C06412=1077.433,-51.002,442.673,173.411,20.692,153.617
C06413=1077.439,-50.753,442.661,173.412,20.694,153.617
C06414=1077.446,-50.504,442.649,173.414,20.696,153.617
C06415=1077.451,-50.254,442.637,173.415,20.698,153.617
C06416=1077.456,-50.004,442.625,173.416,20.700,153.617
C06417=1077.464,-49.729,442.612,173.418,20.702,153.618
C06418=1077.470,-49.454,442.599,173.420,20.704,153.618
C06419=1077.476,-49.180,442.586,173.421,20.706,153.618
C06420=1077.483,-48.905,442.571,173.422,20.708,153.618
C06421=1077.489,-48.656,442.561,173.424,20.709,153.618
C06422=1077.495,-48.406,442.548,173.425,20.711,153.618
C06423=1077.501,-48.156,442.535,173.427,20.714,153.618
C06424=1077.507,-47.907,442.524,173.429,20.716,153.618
C06425=1077.513,-47.657,442.511,173.430,20.718,153.619
C06426=1077.519,-47.407,442.500,173.431,20.720,153.619
C06427=1077.524,-47.158,442.488,173.433,20.722,153.619
C06428=1077.530,-46.908,442.475,173.434,20.723,153.619
C06429=1077.537,-46.658,442.463,173.436,20.725,153.619
C06430=1077.542,-46.409,442.451,173.437,20.727,153.619
C06431=1077.548,-46.159,442.439,173.438,20.729,153.619
C06432=1077.555,-45.910,442.427,173.440,20.732,153.620
C06433=1077.560,-45.660,442.415,173.442,20.734,153.620
C06434=1077.566,-45.410,442.403,173.443,20.735,153.620
C06435=1077.572,-45.160,442.391,173.444,20.737,153.620
C06436=1077.578,-44.911,442.379,173.446,20.739,153.620
C06437=1077.584,-44.662,442.367,173.447,20.741,153.620
C06438=1077.590,-44.412,442.354,173.448,20.743,153.620
C06439=1077.596,-44.162,442.341,173.450,20.745,153.621
C06440=1077.602,-43.913,442.330,173.451,20.747,153.621
C06441=1077.608,-43.663,442.317,173.453,20.749,153.621
C06442=1077.614,-43.413,442.305,173.455,20.751,153.621
C06443=1077.621,-43.164,442.293,173.456,20.753,153.621
C06444=1077.626,-42.914,442.281,173.457,20.755,153.621
C06445=1077.632,-42.665,442.268,173.458,20.757,153.621
C06446=1077.639,-42.415,442.256,173.460,20.759,153.622
C06447=1077.645,-42.165,442.244,173.461,20.761,153.622
C06448=1077.650,-41.916,442.231,173.463,20.763,153.622
C06449=1077.656,-41.666,442.219,173.465,20.765,153.622
C06450=1077.662,-41.416,442.207,173.466,20.767,153.622
C06451=1077.668,-41.167,442.194,173.467,20.769,153.622
C06452=1077.674,-40.917,442.182,173.469,20.771,153.622
C06453=1077.680,-40.668,442.170,173.470,20.773,153.623
C06454=1077.686,-40.418,442.158,173.471,20.775,153.623
C06455=1077.692,-40.168,442.145,173.473,20.777,153.623
C06456=1077.699,-39.918,442.133,173.474,20.779,153.623
C06457=1077.704,-39.669,442.121,173.475,20.781,153.623
C06458=1077.710,-39.419,442.108,173.478,20.783,153.623
C06459=1077.716,-39.170,442.096,173.479,20.785,153.623
C06460=1077.722,-38.920,442.084,173.480,20.787,153.624
C06461=1077.728,-38.670,442.071,173.482,20.789,153.624
C06462=1077.734,-38.421,442.059,173.483,20.791,153.624
C06463=1077.740,-38.171,442.046,173.484,20.793,153.624
C06464=1077.746,-37.921,442.034,173.486,20.795,153.624
C06465=1077.751,-37.671,442.021,173.488,20.797,153.624
C06466=1077.758,-37.422,442.009,173.489,20.799,153.624
C06467=1077.764,-37.173,441.997,173.490,20.802,153.625
C06468=1077.770,-36.923,441.984,173.491,20.803,153.625
C06469=1077.775,-36.673,441.971,173.493,20.805,153.625
C06470=1077.781,-36.423,441.959,173.494,20.807,153.625
C06471=1077.787,-36.174,441.947,173.495,20.809,153.625
C06472=1077.793,-35.924,441.934,173.497,20.811,153.626
C06473=1077.799,-35.675,441.921,173.499,20.814,153.626
C06474=1077.805,-35.425,441.908,173.500,20.816,153.626
C06475=1077.811,-35.175,441.896,173.502,20.818,153.626
C06476=1077.817,-34.925,441.883,173.503,20.820,153.626
C06477=1077.823,-34.677,441.872,173.504,20.822,153.626
C06478=1077.829,-34.427,441.858,173.505,20.824,153.627
C06479=1077.835,-34.177,441.846,173.507,20.826,153.627
C06480=1077.841,-33.928,441.833,173.509,20.828,153.627
C06481=1077.847,-33.654,441.819,173.510,20.831,153.627
C06482=1077.853,-33.379,441.806,173.511,20.833,153.627
C06483=1077.860,-33.104,441.792,173.514,20.835,153.627
C06484=1077.866,-32.830,441.777,173.515,20.837,153.628
C06485=1077.873,-32.580,441.765,173.516,20.839,153.628
C06486=1077.879,-32.331,441.752,173.518,20.841,153.628
C06487=1077.885,-32.081,441.740,173.519,20.843,153.628
C06488=1077.890,-31.832,441.727,173.521,20.846,153.628
C06489=1077.896,-31.582,441.715,173.522,20.848,153.628
C06490=1077.902,-31.333,441.702,173.523,20.850,153.629
C06491=1077.908,-31.083,441.689,173.525,20.852,153.629
C06492=1077.914,-30.833,441.676,173.526,20.854,153.629
C06493=1077.920,-30.584,441.663,173.527,20.856,153.629
C06494=1077.926,-30.334,441.651,173.529,20.858,153.629
C06495=1077.932,-30.084,441.638,173.531,20.860,153.629
C06496=1077.938,-29.835,441.625,173.532,20.862,153.630
C06497=1077.944,-29.585,441.612,173.534,20.864,153.630
C06498=1077.950,-29.336,441.600,173.535,20.867,153.630
C06499=1077.956,-29.086,441.587,173.536,20.869,153.630
C06500=1077.962,-28.837,441.574,173.537,20.871,153.630
C06501=1077.968,-28.587,441.562,173.539,20.873,153.631
C06502=1077.974,-28.337,441.548,173.541,20.875,153.631
C06503=1077.980,-28.088,441.536,173.542,20.877,153.631
C06504=1077.986,-27.838,441.523,173.543,20.879,153.631
C06505=1077.992,-27.588,441.510,173.545,20.881,153.631
C06506=1077.998,-27.338,441.498,173.546,20.883,153.631
C06507=1078.004,-27.089,441.484,173.547,20.885,153.631
C06508=1078.010,-26.839,441.472,173.548,20.887,153.632
C06509=1078.016,-26.590,441.458,173.551,20.890,153.632
C06510=1078.022,-26.340,441.446,173.552,20.892,153.632
C06511=1078.027,-26.091,441.432,173.553,20.894,153.632
C06512=1078.033,-25.841,441.419,173.555,20.896,153.632
C06513=1078.040,-25.591,441.406,173.556,20.898,153.633
C06514=1078.045,-25.342,441.394,173.557,20.900,153.633
C06515=1078.051,-25.092,441.381,173.559,20.903,153.633
C06516=1078.056,-24.843,441.368,173.561,20.905,153.633
C06517=1078.062,-24.593,441.355,173.562,20.906,153.633
C06518=1078.068,-24.344,441.342,173.563,20.909,153.634
C06519=1078.074,-24.094,441.329,173.564,20.911,153.634
C06520=1078.081,-23.845,441.316,173.566,20.913,153.634
C06521=1078.086,-23.594,441.303,173.568,20.915,153.634
C06522=1078.092,-23.345,441.290,173.569,20.918,153.634
C06523=1078.098,-23.096,441.276,173.570,20.920,153.634
C06524=1078.104,-22.846,441.264,173.572,20.922,153.635
C06525=1078.110,-22.597,441.250,173.573,20.924,153.635
C06526=1078.115,-22.346,441.237,173.574,20.926,153.635
C06527=1078.122,-22.097,441.224,173.576,20.929,153.635
C06528=1078.128,-21.847,441.211,173.578,20.931,153.635
C06529=1078.134,-21.598,441.198,173.579,20.933,153.636
C06530=1078.139,-21.348,441.184,173.580,20.935,153.636
C06531=1078.145,-21.099,441.172,173.581,20.937,153.636
C06532=1078.151,-20.849,441.158,173.583,20.939,153.636
C06533=1078.157,-20.599,441.146,173.585,20.941,153.636
C06534=1078.163,-20.350,441.132,173.586,20.943,153.636
C06535=1078.169,-20.101,441.119,173.587,20.946,153.637
C06536=1078.175,-19.851,441.106,173.589,20.948,153.637
C06537=1078.181,-19.601,441.093,173.590,20.950,153.637
C06538=1078.186,-19.351,441.080,173.591,20.952,153.637
C06539=1078.192,-19.102,441.067,173.593,20.955,153.638
C06540=1078.199,-18.853,441.053,173.594,20.957,153.638
C06541=1078.205,-18.603,441.041,173.596,20.959,153.638
C06542=1078.210,-18.353,441.027,173.597,20.961,153.638
C06543=1078.216,-18.104,441.014,173.598,20.963,153.638
C06544=1078.222,-17.855,441.000,173.600,20.965,153.638
C06545=1078.228,-17.579,440.986,173.602,20.968,153.639
C06546=1078.235,-17.303,440.971,173.603,20.970,153.639
C06547=1078.242,-17.029,440.957,173.605,20.973,153.639
C06548=1078.249,-16.754,440.942,173.606,20.975,153.639
C06549=1078.255,-16.504,440.929,173.607,20.977,153.639
C06550=1078.260,-16.254,440.915,173.609,20.979,153.640
C06551=1078.266,-16.005,440.902,173.610,20.981,153.640
C06552=1078.273,-15.756,440.889,173.612,20.984,153.640
C06553=1078.278,-15.506,440.875,173.613,20.986,153.640
C06554=1078.284,-15.256,440.862,173.615,20.988,153.640
C06555=1078.290,-15.007,440.849,173.616,20.990,153.641
C06556=1078.296,-14.757,440.835,173.617,20.992,153.641
C06557=1078.303,-14.507,440.822,173.619,20.995,153.641
C06558=1078.308,-14.257,440.809,173.621,20.997,153.641
C06559=1078.314,-14.008,440.795,173.622,20.999,153.641
C06560=1078.319,-13.758,440.781,173.623,21.001,153.642
C06561=1078.326,-13.509,440.768,173.624,21.004,153.642
C06562=1078.331,-13.259,440.754,173.626,21.006,153.642
C06563=1078.337,-13.010,440.741,173.628,21.008,153.642
C06564=1078.343,-12.760,440.728,173.629,21.011,153.642
C06565=1078.349,-12.511,440.715,173.630,21.013,153.643
C06566=1078.355,-12.262,440.701,173.632,21.014,153.643
C06567=1078.360,-12.012,440.687,173.633,21.017,153.643
C06568=1078.367,-11.763,440.674,173.634,21.019,153.643
C06569=1078.373,-11.512,440.660,173.636,21.021,153.643
C06570=1078.379,-11.263,440.647,173.637,21.024,153.644
C06571=1078.384,-11.013,440.634,173.639,21.026,153.644
C06572=1078.390,-10.763,440.620,173.640,21.028,153.644
C06573=1078.396,-10.514,440.606,173.641,21.030,153.644
C06574=1078.401,-10.265,440.593,173.643,21.033,153.644
C06575=1078.407,-10.015,440.579,173.645,21.035,153.645
C06576=1078.413,-9.766,440.565,173.646,21.037,153.645
C06577=1078.420,-9.516,440.552,173.647,21.039,153.645
C06578=1078.425,-9.266,440.538,173.648,21.042,153.645
C06579=1078.431,-9.017,440.525,173.650,21.044,153.646
C06580=1078.437,-8.767,440.511,173.652,21.046,153.646
C06581=1078.443,-8.518,440.497,173.653,21.049,153.646
C06582=1078.449,-8.268,440.484,173.654,21.050,153.646
C06583=1078.455,-8.019,440.470,173.655,21.052,153.646
C06584=1078.461,-7.769,440.456,173.657,21.055,153.647
C06585=1078.467,-7.520,440.443,173.659,21.057,153.647
C06586=1078.473,-7.270,440.429,173.660,21.059,153.647
C06587=1078.478,-7.021,440.415,173.661,21.062,153.647
C06588=1078.484,-6.771,440.402,173.663,21.064,153.647
C06589=1078.490,-6.521,440.388,173.664,21.066,153.648
C06590=1078.497,-6.272,440.374,173.666,21.069,153.648
C06591=1078.502,-6.022,440.360,173.667,21.071,153.648
C06592=1078.508,-5.773,440.347,173.668,21.073,153.648
C06593=1078.514,-5.523,440.333,173.670,21.075,153.648
C06594=1078.520,-5.273,440.319,173.671,21.077,153.649
C06595=1078.526,-5.024,440.306,173.673,21.080,153.649
C06596=1078.531,-4.774,440.292,173.674,21.082,153.649
C06597=1078.538,-4.525,440.279,173.676,21.084,153.649
C06598=1078.544,-4.275,440.264,173.677,21.086,153.649
C06599=1078.550,-4.026,440.251,173.678,21.088,153.650
C06600=1078.556,-3.776,440.237,173.680,21.091,153.650
C06601=1078.561,-3.527,440.223,173.681,21.093,153.650
C06602=1078.568,-3.277,440.209,173.683,21.095,153.650
C06603=1078.574,-3.027,440.195,173.684,21.098,153.651
C06604=1078.579,-2.778,440.181,173.685,21.100,153.651
C06605=1078.584,-2.528,440.168,173.687,21.103,153.651
C06606=1078.590,-2.279,440.153,173.688,21.105,153.651
C06607=1078.596,-2.030,440.140,173.690,21.107,153.651
C06608=1078.603,-1.780,440.125,173.691,21.109,153.652
C06609=1078.608,-1.503,440.110,173.693,21.112,153.652
C06610=1078.615,-1.226,440.094,173.694,21.115,153.652
C06611=1078.621,-0.949,440.079,173.695,21.116,153.652
C06612=1078.628,-0.672,440.064,173.697,21.119,153.653
C06613=1078.633,-0.423,440.049,173.698,21.122,153.653
C06614=1078.640,-0.174,440.036,173.700,21.124,153.653
C06615=1078.646,0.076,440.022,173.702,21.127,153.653
C06616=1078.651,0.326,440.008,173.703,21.129,153.653
C06617=1078.657,0.576,439.994,173.704,21.131,153.654
C06618=1078.662,0.825,439.979,173.706,21.133,153.654
C06619=1078.668,1.074,439.965,173.707,21.136,153.654
C06620=1078.675,1.324,439.952,173.709,21.138,153.654
C06621=1078.680,1.573,439.937,173.710,21.141,153.655
C06622=1078.686,1.823,439.923,173.711,21.143,153.655
C06623=1078.691,2.072,439.909,173.713,21.145,153.655
C06624=1078.697,2.322,439.895,173.714,21.147,153.655
C06625=1078.703,2.571,439.881,173.716,21.149,153.655
C06626=1078.709,2.821,439.867,173.717,21.152,153.656
C06627=1078.715,3.071,439.852,173.719,21.154,153.656
C06628=1078.721,3.320,439.839,173.720,21.156,153.656
C06629=1078.727,3.569,439.825,173.721,21.158,153.656
C06630=1078.732,3.819,439.811,173.723,21.161,153.657
C06631=1078.739,4.069,439.796,173.724,21.163,153.657
C06632=1078.744,4.318,439.782,173.725,21.166,153.657
C06633=1078.750,4.568,439.768,173.727,21.168,153.657
C06634=1078.756,4.817,439.753,173.728,21.170,153.658
C06635=1078.761,5.067,439.739,173.730,21.173,153.658
C06636=1078.767,5.316,439.725,173.731,21.175,153.658
C06637=1078.773,5.566,439.710,173.733,21.177,153.658
C06638=1078.780,5.816,439.697,173.734,21.180,153.658
C06639=1078.785,6.065,439.683,173.736,21.182,153.659
C06640=1078.791,6.315,439.668,173.737,21.184,153.659
C06641=1078.797,6.564,439.654,173.738,21.186,153.659
C06642=1078.803,6.813,439.640,173.739,21.189,153.659
C06643=1078.809,7.064,439.626,173.741,21.191,153.659
C06644=1078.815,7.313,439.611,173.743,21.193,153.660
C06645=1078.820,7.562,439.597,173.744,21.196,153.660
C06646=1078.826,7.812,439.582,173.745,21.198,153.660
C06647=1078.832,8.061,439.568,173.747,21.200,153.660
C06648=1078.838,8.310,439.554,173.749,21.203,153.660
C06649=1078.844,8.561,439.540,173.750,21.205,153.661
C06650=1078.850,8.810,439.525,173.751,21.207,153.661
C06651=1078.856,9.060,439.511,173.752,21.209,153.661
C06652=1078.861,9.309,439.496,173.754,21.211,153.661
C06653=1078.867,9.558,439.482,173.756,21.214,153.662
C06654=1078.874,9.808,439.468,173.757,21.216,153.662
C06655=1078.879,10.057,439.454,173.758,21.219,153.662
C06656=1078.886,10.307,439.439,173.760,21.221,153.662
C06657=1078.891,10.557,439.425,173.761,21.223,153.663
C06658=1078.897,10.805,439.411,173.763,21.226,153.663
C06659=1078.903,11.055,439.396,173.764,21.228,153.663
C06660=1078.909,11.305,439.382,173.765,21.230,153.663
C06661=1078.915,11.554,439.367,173.767,21.232,153.663
C06662=1078.921,11.804,439.353,173.769,21.235,153.664
C06663=1078.927,12.054,439.338,173.770,21.237,153.664
C06664=1078.933,12.303,439.324,173.771,21.239,153.664
C06665=1078.939,12.553,439.309,173.772,21.241,153.664
C06666=1078.945,12.802,439.295,173.774,21.244,153.665
C06667=1078.951,13.052,439.281,173.776,21.246,153.665
C06668=1078.957,13.301,439.266,173.777,21.249,153.665
C06669=1078.962,13.550,439.251,173.778,21.251,153.665
C06670=1078.969,13.800,439.237,173.780,21.253,153.665
C06671=1078.974,14.049,439.223,173.782,21.256,153.666
C06672=1078.981,14.299,439.208,173.783,21.258,153.666
C06673=1078.987,14.578,439.192,173.784,21.260,153.666
C06674=1078.994,14.857,439.175,173.786,21.263,153.666
C06675=1079.000,15.135,439.159,173.787,21.265,153.667
C06676=1079.006,15.414,439.142,173.789,21.268,153.667
C06677=1079.012,15.664,439.128,173.791,21.270,153.667
C06678=1079.018,15.913,439.113,173.792,21.273,153.667
C06679=1079.023,16.162,439.098,173.793,21.275,153.668
C06680=1079.029,16.413,439.084,173.795,21.278,153.668
C06681=1079.035,16.662,439.070,173.796,21.280,153.668
C06682=1079.042,16.911,439.055,173.798,21.282,153.668
C06683=1079.047,17.160,439.040,173.799,21.284,153.668
C06684=1079.053,17.411,439.025,173.801,21.287,153.669
C06685=1079.058,17.660,439.011,173.802,21.289,153.669
C06686=1079.065,17.909,438.996,173.803,21.291,153.669
C06687=1079.071,18.158,438.981,173.804,21.294,153.669
C06688=1079.077,18.408,438.966,173.807,21.296,153.670
C06689=1079.082,18.658,438.952,173.808,21.299,153.670
C06690=1079.088,18.908,438.937,173.809,21.301,153.670
C06691=1079.094,19.157,438.922,173.810,21.303,153.670
C06692=1079.100,19.406,438.907,173.813,21.306,153.670
C06693=1079.105,19.655,438.892,173.814,21.308,153.671
C06694=1079.111,19.906,438.878,173.815,21.310,153.671
C06695=1079.117,20.155,438.863,173.816,21.313,153.671
C06696=1079.124,20.404,438.848,173.818,21.315,153.671
C06697=1079.129,20.654,438.833,173.819,21.317,153.672
C06698=1079.135,20.903,438.818,173.821,21.319,153.672
C06699=1079.141,21.152,438.804,173.822,21.322,153.672
C06700=1079.146,21.402,438.788,173.823,21.324,153.672
C06701=1079.152,21.651,438.773,173.825,21.327,153.673
C06702=1079.158,21.901,438.759,173.826,21.329,153.673
C06703=1079.163,22.151,438.744,173.828,21.331,153.673
C06704=1079.170,22.400,438.729,173.829,21.334,153.673
C06705=1079.175,22.649,438.714,173.831,21.336,153.673
C06706=1079.181,22.899,438.699,173.832,21.339,153.674
C06707=1079.188,23.149,438.684,173.834,21.340,153.674
C06708=1079.193,23.398,438.669,173.835,21.343,153.674
C06709=1079.199,23.648,438.654,173.837,21.345,153.674
C06710=1079.205,23.897,438.639,173.838,21.348,153.675
C06711=1079.210,24.147,438.624,173.839,21.350,153.675
C06712=1079.216,24.396,438.609,173.841,21.352,153.675
C06713=1079.223,24.645,438.594,173.843,21.355,153.675
C06714=1079.228,24.895,438.579,173.844,21.357,153.676
C06715=1079.234,25.144,438.564,173.845,21.360,153.676
C06716=1079.240,25.394,438.549,173.846,21.362,153.676
C06717=1079.245,25.643,438.534,173.848,21.364,153.676
C06718=1079.252,25.893,438.519,173.850,21.366,153.676
C06719=1079.257,26.142,438.504,173.851,21.369,153.677
C06720=1079.263,26.392,438.489,173.852,21.371,153.677
C06721=1079.269,26.642,438.473,173.854,21.374,153.677
C06722=1079.275,26.891,438.459,173.856,21.376,153.677
C06723=1079.281,27.140,438.444,173.857,21.378,153.678
C06724=1079.286,27.390,438.429,173.858,21.380,153.678
C06725=1079.292,27.639,438.414,173.860,21.383,153.678
C06726=1079.298,27.889,438.398,173.861,21.386,153.678
C06727=1079.304,28.138,438.384,173.863,21.387,153.679
C06728=1079.310,28.388,438.367,173.865,21.390,153.679
C06729=1079.316,28.637,438.353,173.866,21.392,153.679
C06730=1079.321,28.887,438.337,173.867,21.395,153.679
C06731=1079.328,29.136,438.322,173.868,21.397,153.679
C06732=1079.333,29.385,438.307,173.871,21.400,153.680
C06733=1079.339,29.635,438.292,173.872,21.402,153.680
C06734=1079.345,29.885,438.277,173.873,21.404,153.680
C06735=1079.350,30.134,438.262,173.874,21.407,153.680
C06736=1079.356,30.383,438.246,173.876,21.409,153.681
C06737=1079.362,30.663,438.229,173.877,21.411,153.681
C06738=1079.369,30.944,438.211,173.880,21.414,153.681
C06739=1079.376,31.224,438.194,173.881,21.417,153.681
C06740=1079.382,31.504,438.177,173.883,21.420,153.682
C06741=1079.388,31.754,438.162,173.884,21.422,153.682
C06742=1079.393,32.003,438.147,173.885,21.424,153.682
C06743=1079.400,32.253,438.132,173.887,21.427,153.682
C06744=1079.405,32.502,438.116,173.889,21.429,153.683
C06745=1079.411,32.751,438.100,173.890,21.432,153.683
C06746=1079.417,33.001,438.085,173.891,21.433,153.683
C06747=1079.423,33.251,438.070,173.893,21.436,153.683
C06748=1079.428,33.500,438.055,173.894,21.438,153.683
C06749=1079.434,33.749,438.039,173.896,21.441,153.684
C06750=1079.440,33.999,438.024,173.897,21.443,153.684
C06751=1079.446,34.249,438.009,173.899,21.446,153.684
C06752=1079.452,34.497,437.993,173.900,21.448,153.684
C06753=1079.457,34.747,437.977,173.901,21.450,153.685
C06754=1079.464,34.997,437.962,173.903,21.453,153.685
C06755=1079.469,35.246,437.947,173.905,21.455,153.685
C06756=1079.475,35.496,437.931,173.906,21.457,153.685
C06757=1079.481,35.745,437.916,173.907,21.459,153.686
C06758=1079.486,35.994,437.901,173.909,21.462,153.686
C06759=1079.493,36.244,437.885,173.911,21.464,153.686
C06760=1079.499,36.493,437.869,173.912,21.467,153.686
C06761=1079.504,36.743,437.853,173.913,21.469,153.687
C06762=1079.510,36.992,437.839,173.915,21.472,153.687
C06763=1079.516,37.242,437.823,173.917,21.473,153.687
C06764=1079.522,37.491,437.807,173.918,21.476,153.687
C06765=1079.528,37.741,437.792,173.920,21.478,153.687
C06766=1079.533,37.990,437.777,173.921,21.481,153.688
C06767=1079.539,38.239,437.760,173.922,21.483,153.688
C06768=1079.545,38.489,437.745,173.924,21.485,153.688
C06769=1079.551,38.739,437.729,173.926,21.488,153.688
C06770=1079.557,38.988,437.714,173.927,21.490,153.689
C06771=1079.563,39.237,437.698,173.928,21.493,153.689
C06772=1079.568,39.487,437.682,173.930,21.495,153.689
C06773=1079.574,39.736,437.666,173.931,21.497,153.689
C06774=1079.579,39.986,437.651,173.933,21.500,153.690
C06775=1079.585,40.236,437.635,173.934,21.502,153.690
C06776=1079.592,40.485,437.620,173.936,21.505,153.690
C06777=1079.597,40.734,437.604,173.937,21.507,153.690
C06778=1079.603,40.983,437.588,173.938,21.509,153.691
C06779=1079.608,41.233,437.573,173.941,21.512,153.691
C06780=1079.614,41.483,437.556,173.942,21.514,153.691
C06781=1079.619,41.732,437.541,173.943,21.516,153.691
C06782=1079.626,41.981,437.526,173.944,21.518,153.691
C06783=1079.632,42.230,437.509,173.946,21.521,153.692
C06784=1079.637,42.480,437.494,173.948,21.523,153.692
C06785=1079.643,42.729,437.478,173.949,21.526,153.692
C06786=1079.648,42.979,437.462,173.951,21.528,153.692
C06787=1079.654,43.228,437.446,173.952,21.531,153.693
C06788=1079.660,43.478,437.431,173.954,21.533,153.693
C06789=1079.666,43.727,437.414,173.956,21.535,153.693
C06790=1079.672,43.977,437.398,173.957,21.537,153.693
C06791=1079.677,44.226,437.383,173.958,21.540,153.693
C06792=1079.683,44.475,437.367,173.959,21.542,153.694
C06793=1079.689,44.725,437.351,173.962,21.545,153.694
C06794=1079.695,44.975,437.335,173.963,21.547,153.694
C06795=1079.700,45.223,437.319,173.964,21.550,153.695
C06796=1079.706,45.473,437.303,173.966,21.552,153.695
C06797=1079.712,45.723,437.287,173.967,21.554,153.695
C06798=1079.717,45.972,437.271,173.969,21.556,153.695
C06799=1079.722,46.221,437.256,173.971,21.559,153.695
C06800=1079.728,46.471,437.239,173.972,21.562,153.696
C06801=1079.735,46.751,437.221,173.973,21.564,153.696
C06802=1079.741,47.031,437.203,173.975,21.567,153.696
C06803=1079.748,47.311,437.186,173.977,21.570,153.696
C06804=1079.754,47.592,437.167,173.978,21.572,153.697
C06805=1079.760,47.841,437.151,173.979,21.574,153.697
C06806=1079.765,48.091,437.136,173.982,21.577,153.697
C06807=1079.771,48.340,437.120,173.983,21.579,153.697
C06808=1079.777,48.589,437.103,173.984,21.582,153.698
C06809=1079.783,48.839,437.087,173.986,21.584,153.698
C06810=1079.789,49.089,437.071,173.987,21.587,153.698
C06811=1079.793,49.338,437.055,173.989,21.589,153.698
C06812=1079.799,49.587,437.039,173.991,21.591,153.699
C06813=1079.805,49.836,437.022,173.992,21.594,153.699
C06814=1079.811,50.086,437.007,173.993,21.596,153.699
C06815=1079.817,50.336,436.991,173.995,21.599,153.699
C06816=1079.823,50.585,436.974,173.997,21.601,153.699
C06817=1079.829,50.834,436.958,173.998,21.603,153.700
C06818=1079.834,51.083,436.942,174.000,21.606,153.700
C06819=1079.839,51.333,436.925,174.001,21.608,153.700
C06820=1079.845,51.583,436.910,174.002,21.610,153.700
C06821=1079.851,51.832,436.894,174.004,21.612,153.701
C06822=1079.857,52.081,436.877,174.006,21.615,153.701
C06823=1079.863,52.331,436.861,174.007,21.617,153.701
C06824=1079.869,52.580,436.845,174.008,21.620,153.701
C06825=1079.875,52.829,436.829,174.011,21.622,153.702
C06826=1079.880,53.079,436.812,174.012,21.625,153.702
C06827=1079.886,53.328,436.795,174.013,21.626,153.702
C06828=1079.891,53.578,436.780,174.015,21.629,153.702
C06829=1079.897,53.827,436.764,174.016,21.631,153.702
C06830=1079.903,54.076,436.748,174.018,21.634,153.703
C06831=1079.909,54.326,436.732,174.020,21.636,153.703
C06832=1079.914,54.575,436.715,174.021,21.639,153.703
C06833=1079.920,54.825,436.698,174.022,21.641,153.703
C06834=1079.926,55.074,436.682,174.024,21.643,153.704
C06835=1079.932,55.323,436.666,174.026,21.645,153.704
C06836=1079.938,55.573,436.650,174.027,21.648,153.704
C06837=1079.944,55.822,436.633,174.029,21.650,153.704
C06838=1079.949,56.072,436.617,174.030,21.653,153.705
C06839=1079.955,56.321,436.600,174.032,21.655,153.705
C06840=1079.961,56.570,436.584,174.034,21.657,153.705
C06841=1079.967,56.820,436.568,174.035,21.659,153.705
C06842=1079.973,57.069,436.552,174.036,21.662,153.705
C06843=1079.978,57.319,436.535,174.038,21.664,153.706
C06844=1079.984,57.568,436.518,174.040,21.667,153.706
C06845=1079.990,57.817,436.502,174.041,21.669,153.706
C06846=1079.996,58.067,436.486,174.043,21.672,153.706
C06847=1080.002,58.316,436.470,174.044,21.673,153.706
C06848=1080.007,58.566,436.453,174.046,21.676,153.707
C06849=1080.013,58.815,436.437,174.048,21.678,153.707
C06850=1080.019,59.064,436.420,174.049,21.680,153.707
C06851=1080.025,59.314,436.404,174.050,21.683,153.707
C06852=1080.030,59.563,436.386,174.053,21.685,153.707
C06853=1080.036,59.812,436.370,174.054,21.687,153.708
C06854=1080.042,60.062,436.354,174.055,21.689,153.708
C06855=1080.048,60.311,436.338,174.057,21.692,153.708
C06856=1080.053,60.561,436.321,174.058,21.694,153.708
C06857=1080.059,60.810,436.305,174.060,21.697,153.709
C06858=1080.066,61.060,436.288,174.062,21.699,153.709
C06859=1080.072,61.309,436.271,174.063,21.701,153.709
C06860=1080.077,61.558,436.254,174.064,21.703,153.709
C06861=1080.083,61.808,436.238,174.067,21.706,153.709
C06862=1080.089,62.057,436.222,174.068,21.708,153.710
C06863=1080.095,62.306,436.205,174.069,21.710,153.710
C06864=1080.100,62.556,436.189,174.071,21.713,153.710
C06865=1080.108,62.836,436.170,174.073,21.715,153.710
C06866=1080.114,63.115,436.151,174.075,21.718,153.711
C06867=1080.121,63.395,436.132,174.077,21.720,153.711
C06868=1080.127,63.675,436.114,174.078,21.723,153.711
C06869=1080.133,63.924,436.097,174.080,21.725,153.711
C06870=1080.139,64.175,436.080,174.081,21.728,153.711
C06871=1080.145,64.424,436.064,174.083,21.730,153.712
C06872=1080.151,64.673,436.047,174.085,21.732,153.712
C06873=1080.157,64.922,436.030,174.086,21.734,153.712
C06874=1080.162,65.172,436.014,174.087,21.737,153.712
C06875=1080.168,65.421,435.997,174.090,21.739,153.712
C06876=1080.174,65.671,435.980,174.091,21.742,153.713
C06877=1080.179,65.920,435.963,174.092,21.744,153.713
C06878=1080.185,66.169,435.947,174.094,21.746,153.713
C06879=1080.190,66.419,435.930,174.096,21.748,153.713
C06880=1080.197,66.667,435.913,174.097,21.750,153.714
C06881=1080.202,66.918,435.896,174.099,21.753,153.714
C06882=1080.208,67.167,435.879,174.100,21.755,153.714
C06883=1080.214,67.416,435.862,174.102,21.758,153.714
C06884=1080.220,67.666,435.846,174.104,21.760,153.714
C06885=1080.225,67.915,435.828,174.105,21.762,153.715
C06886=1080.231,68.164,435.812,174.107,21.765,153.715
C06887=1080.237,68.414,435.795,174.109,21.767,153.715
C06888=1080.243,68.662,435.778,174.110,21.769,153.715
C06889=1080.249,68.913,435.761,174.112,21.771,153.715
C06890=1080.254,69.162,435.743,174.113,21.774,153.716
C06891=1080.260,69.411,435.727,174.115,21.776,153.716
C06892=1080.265,69.661,435.710,174.117,21.779,153.716
C06893=1080.272,69.909,435.693,174.118,21.781,153.716
C06894=1080.277,70.159,435.676,174.119,21.783,153.717
C06895=1080.283,70.408,435.659,174.121,21.785,153.717
C06896=1080.289,70.658,435.642,174.123,21.787,153.717
C06897=1080.294,70.907,435.624,174.125,21.790,153.717
C06898=1080.300,71.157,435.608,174.126,21.792,153.717
C06899=1080.306,71.406,435.591,174.127,21.795,153.718
C06900=1080.311,71.655,435.574,174.130,21.797,153.718
C06901=1080.317,71.904,435.557,174.131,21.799,153.718
C06902=1080.322,72.154,435.540,174.132,21.801,153.718
C06903=1080.329,72.403,435.522,174.134,21.804,153.718
C06904=1080.335,72.653,435.506,174.135,21.806,153.719
C06905=1080.340,72.902,435.488,174.138,21.809,153.719
C06906=1080.345,73.151,435.471,174.139,21.811,153.719
C06907=1080.352,73.400,435.454,174.140,21.813,153.719
C06908=1080.357,73.651,435.437,174.142,21.816,153.720
C06909=1080.363,73.900,435.420,174.144,21.818,153.720
C06910=1080.368,74.149,435.402,174.145,21.820,153.720
C06911=1080.374,74.398,435.386,174.147,21.823,153.720
C06912=1080.380,74.647,435.368,174.148,21.824,153.720
C06913=1080.386,74.897,435.351,174.151,21.827,153.721
C06914=1080.392,75.146,435.334,174.152,21.829,153.721
C06915=1080.397,75.395,435.316,174.153,21.831,153.721
C06916=1080.403,75.645,435.300,174.155,21.834,153.721
C06917=1080.408,75.894,435.282,174.157,21.836,153.721
C06918=1080.415,76.143,435.265,174.158,21.838,153.722
C06919=1080.420,76.393,435.248,174.160,21.841,153.722
C06920=1080.426,76.642,435.230,174.162,21.843,153.722
C06921=1080.431,76.891,435.213,174.164,21.846,153.722
C06922=1080.438,77.141,435.196,174.165,21.848,153.723
C06923=1080.443,77.390,435.178,174.166,21.849,153.723
C06924=1080.449,77.639,435.161,174.168,21.852,153.723
C06925=1080.454,77.889,435.144,174.170,21.854,153.723
C06926=1080.461,78.138,435.127,174.172,21.857,153.723
C06927=1080.466,78.387,435.109,174.173,21.859,153.724
C06928=1080.472,78.636,435.092,174.175,21.861,153.724
C06929=1080.478,78.916,435.073,174.177,21.864,153.724
C06930=1080.485,79.197,435.052,174.179,21.867,153.724
C06931=1080.491,79.477,435.033,174.180,21.869,153.724
C06932=1080.498,79.756,435.014,174.182,21.872,153.725
C06933=1080.503,80.005,434.996,174.184,21.874,153.725
C06934=1080.508,80.255,434.979,174.185,21.876,153.725
C06935=1080.514,80.505,434.961,174.187,21.878,153.725
C06936=1080.520,80.754,434.944,174.189,21.881,153.726
C06937=1080.526,81.003,434.926,174.190,21.883,153.726
C06938=1080.531,81.252,434.909,174.193,21.885,153.726
C06939=1080.537,81.502,434.891,174.194,21.888,153.726
C06940=1080.542,81.751,434.874,174.195,21.890,153.726
C06941=1080.548,82.000,434.856,174.197,21.893,153.727
C06942=1080.554,82.250,434.838,174.199,21.895,153.727
C06943=1080.560,82.499,434.821,174.201,21.897,153.727
C06944=1080.565,82.748,434.803,174.202,21.899,153.727
C06945=1080.571,82.997,434.786,174.203,21.901,153.727
C06946=1080.577,83.247,434.768,174.206,21.904,153.728
C06947=1080.582,83.496,434.751,174.207,21.906,153.728
C06948=1080.587,83.745,434.733,174.209,21.908,153.728
C06949=1080.594,83.995,434.715,174.210,21.910,153.728
C06950=1080.599,84.244,434.698,174.212,21.913,153.728
C06951=1080.605,84.493,434.680,174.214,21.915,153.729
C06952=1080.611,84.743,434.662,174.215,21.917,153.729
C06953=1080.616,84.992,434.645,174.217,21.920,153.729
C06954=1080.622,85.241,434.627,174.219,21.922,153.729
C06955=1080.628,85.491,434.609,174.220,21.924,153.729
C06956=1080.633,85.740,434.592,174.222,21.927,153.730
C06957=1080.639,85.989,434.574,174.223,21.929,153.730
C06958=1080.645,86.239,434.556,174.226,21.931,153.730
C06959=1080.651,86.488,434.539,174.227,21.933,153.730
C06960=1080.657,86.737,434.521,174.229,21.936,153.730
C06961=1080.662,86.986,434.503,174.231,21.938,153.731
C06962=1080.668,87.235,434.485,174.232,21.940,153.731
C06963=1080.674,87.485,434.468,174.234,21.942,153.731
C06964=1080.679,87.734,434.450,174.235,21.944,153.731
C06965=1080.685,87.984,434.432,174.238,21.947,153.731
C06966=1080.691,88.233,434.414,174.239,21.949,153.732
C06967=1080.696,88.482,434.397,174.241,21.952,153.732
C06968=1080.703,88.732,434.379,174.242,21.953,153.732
C06969=1080.708,88.981,434.361,174.244,21.955,153.732
C06970=1080.714,89.231,434.343,174.246,21.958,153.732
C06971=1080.720,89.479,434.325,174.247,21.960,153.732
C06972=1080.726,89.728,434.308,174.249,21.962,153.733
C06973=1080.732,89.978,434.290,174.251,21.964,153.733
C06974=1080.736,90.227,434.272,174.253,21.967,153.733
C06975=1080.743,90.477,434.254,174.254,21.969,153.733
C06976=1080.748,90.726,434.236,174.256,21.971,153.733
C06977=1080.754,90.976,434.218,174.258,21.973,153.734
C06978=1080.760,91.224,434.200,174.259,21.976,153.734
C06979=1080.766,91.474,434.182,174.261,21.978,153.734
C06980=1080.771,91.723,434.164,174.263,21.980,153.734
C06981=1080.776,91.972,434.146,174.265,21.983,153.734
C06982=1080.783,92.222,434.128,174.266,21.985,153.735
C06983=1080.788,92.470,434.110,174.268,21.987,153.735
C06984=1080.794,92.720,434.091,174.270,21.989,153.735
C06985=1080.799,92.970,434.074,174.271,21.992,153.735
C06986=1080.805,93.219,434.056,174.273,21.994,153.735
C06987=1080.811,93.468,434.038,174.275,21.996,153.735
C06988=1080.816,93.717,434.019,174.277,21.999,153.736
C06989=1080.822,93.967,434.002,174.278,22.001,153.736
C06990=1080.828,94.216,433.984,174.280,22.003,153.736
C06991=1080.833,94.466,433.965,174.282,22.005,153.736
C06992=1080.839,94.714,433.947,174.284,22.008,153.737
C06993=1080.845,94.995,433.926,174.285,22.010,153.737
C06994=1080.852,95.274,433.907,174.287,22.013,153.737
C06995=1080.858,95.555,433.887,174.290,22.015,153.737
C06996=1080.864,95.834,433.866,174.292,22.018,153.737
C06997=1080.871,96.083,433.848,174.293,22.020,153.738
C06998=1080.875,96.333,433.829,174.294,22.022,153.738
C06999=1080.882,96.582,433.811,174.297,22.024,153.738
C07000=1080.887,96.831,433.793,174.298,22.026,153.738
C07001=1080.893,97.081,433.775,174.300,22.029,153.738
C07002=1080.898,97.330,433.757,174.301,22.031,153.738
C07003=1080.905,97.579,433.738,174.304,22.033,153.739
C07004=1080.910,97.828,433.720,174.305,22.035,153.739
C07005=1080.916,98.078,433.702,174.307,22.038,153.739
C07006=1080.921,98.327,433.684,174.309,22.040,153.739
C07007=1080.927,98.577,433.666,174.311,22.042,153.739
C07008=1080.933,98.825,433.647,174.312,22.044,153.739
C07009=1080.939,99.075,433.629,174.314,22.046,153.740
C07010=1080.945,99.324,433.610,174.316,22.048,153.740
C07011=1080.950,99.573,433.592,174.317,22.051,153.740
C07012=1080.956,99.822,433.574,174.319,22.053,153.740
C07013=1080.961,100.072,433.556,174.321,22.055,153.740
C07014=1080.968,100.321,433.537,174.323,22.057,153.741
C07015=1080.972,100.570,433.519,174.324,22.059,153.741
C07016=1080.979,100.819,433.500,174.327,22.061,153.741
C07017=1080.985,101.069,433.482,174.328,22.064,153.741
C07018=1080.990,101.318,433.463,174.330,22.066,153.741
C07019=1080.996,101.568,433.445,174.331,22.068,153.741
C07020=1081.001,101.816,433.427,174.334,22.070,153.742
C07021=1081.007,102.066,433.409,174.335,22.072,153.742
C07022=1081.012,102.315,433.390,174.337,22.075,153.742
C07023=1081.018,102.565,433.371,174.339,22.077,153.742
C07024=1081.024,102.813,433.353,174.341,22.079,153.742
C07025=1081.029,103.063,433.334,174.342,22.081,153.743
C07026=1081.035,103.312,433.316,174.344,22.084,153.743
C07027=1081.041,103.561,433.297,174.346,22.086,153.743
C07028=1081.047,103.811,433.279,174.348,22.089,153.743
C07029=1081.052,104.060,433.260,174.349,22.090,153.743
C07030=1081.057,104.309,433.241,174.352,22.093,153.743
C07031=1081.064,104.559,433.223,174.353,22.095,153.744
C07032=1081.069,104.807,433.204,174.355,22.098,153.744
C07033=1081.075,105.057,433.186,174.356,22.099,153.744
C07034=1081.080,105.306,433.167,174.359,22.102,153.744
C07035=1081.086,105.555,433.149,174.360,22.104,153.744
C07036=1081.092,105.805,433.130,174.362,22.106,153.744
C07037=1081.097,106.054,433.111,174.364,22.108,153.745
C07038=1081.103,106.303,433.093,174.365,22.110,153.745
C07039=1081.108,106.552,433.074,174.367,22.113,153.745
C07040=1081.114,106.801,433.056,174.369,22.115,153.745
C07041=1081.120,107.051,433.037,174.371,22.117,153.745
C07042=1081.125,107.300,433.018,174.372,22.119,153.746
C07043=1081.131,107.549,433.000,174.374,22.121,153.746
C07044=1081.137,107.799,432.980,174.376,22.123,153.746
C07045=1081.142,108.048,432.962,174.378,22.125,153.746
C07046=1081.149,108.297,432.943,174.380,22.127,153.746
C07047=1081.154,108.546,432.924,174.382,22.130,153.746
C07048=1081.159,108.795,432.906,174.384,22.132,153.746
C07049=1081.165,109.045,432.887,174.385,22.134,153.747
C07050=1081.171,109.294,432.868,174.388,22.137,153.747
C07051=1081.177,109.542,432.849,174.389,22.139,153.747
C07052=1081.183,109.792,432.830,174.391,22.141,153.747
C07053=1081.188,110.042,432.812,174.393,22.143,153.747
C07054=1081.194,110.291,432.793,174.395,22.145,153.747
C07055=1081.200,110.540,432.774,174.396,22.147,153.748
C07056=1081.205,110.789,432.755,174.398,22.149,153.748
C07057=1081.212,111.069,432.734,174.400,22.151,153.748
C07058=1081.219,111.349,432.713,174.402,22.154,153.748
C07059=1081.224,111.630,432.691,174.404,22.157,153.748
C07060=1081.231,111.909,432.670,174.406,22.159,153.749
C07061=1081.236,112.158,432.651,174.408,22.161,153.749
C07062=1081.243,112.407,432.632,174.410,22.163,153.749
C07063=1081.248,112.657,432.614,174.412,22.165,153.749
C07064=1081.253,112.906,432.595,174.414,22.168,153.749
C07065=1081.259,113.155,432.576,174.416,22.170,153.749
C07066=1081.265,113.405,432.556,174.417,22.172,153.750
C07067=1081.271,113.654,432.538,174.420,22.174,153.750
C07068=1081.276,113.903,432.519,174.421,22.176,153.750
C07069=1081.282,114.152,432.500,174.423,22.179,153.750
C07070=1081.287,114.401,432.480,174.425,22.181,153.750
C07071=1081.293,114.651,432.461,174.427,22.183,153.750
C07072=1081.298,114.900,432.442,174.428,22.185,153.750
C07073=1081.304,115.149,432.423,174.431,22.187,153.751
C07074=1081.310,115.399,432.404,174.432,22.189,153.751
C07075=1081.315,115.647,432.385,174.434,22.191,153.751
C07076=1081.320,115.897,432.366,174.435,22.194,153.751
C07077=1081.326,116.146,432.346,174.438,22.196,153.751
C07078=1081.332,116.396,432.327,174.439,22.198,153.752
C07079=1081.337,116.644,432.308,174.441,22.200,153.752
C07080=1081.343,116.893,432.288,174.444,22.203,153.752
C07081=1081.349,117.143,432.269,174.445,22.205,153.752
C07082=1081.354,117.392,432.250,174.447,22.207,153.752
C07083=1081.359,117.641,432.231,174.449,22.209,153.752
C07084=1081.365,117.890,432.212,174.451,22.211,153.752
C07085=1081.371,118.140,432.192,174.452,22.213,153.753
C07086=1081.376,118.389,432.173,174.455,22.215,153.753
C07087=1081.381,118.638,432.154,174.456,22.218,153.753
C07088=1081.387,118.887,432.135,174.458,22.220,153.753
C07089=1081.393,119.136,432.115,174.459,22.222,153.753
C07090=1081.399,119.385,432.096,174.462,22.224,153.754
C07091=1081.404,119.634,432.077,174.464,22.227,153.754
C07092=1081.410,119.884,432.058,174.465,22.229,153.754
C07093=1081.415,120.133,432.039,174.468,22.231,153.754
C07094=1081.421,120.382,432.019,174.469,22.233,153.754
C07095=1081.427,120.631,431.999,174.471,22.235,153.754
C07096=1081.432,120.880,431.980,174.473,22.237,153.754
C07097=1081.438,121.129,431.961,174.475,22.239,153.755
C07098=1081.443,121.379,431.942,174.477,22.242,153.755
C07099=1081.449,121.628,431.922,174.479,22.244,153.755
C07100=1081.455,121.877,431.903,174.481,22.246,153.755
C07101=1081.461,122.127,431.884,174.482,22.248,153.755
C07102=1081.466,122.376,431.864,174.485,22.250,153.755
C07103=1081.471,122.624,431.844,174.486,22.252,153.756
C07104=1081.477,122.874,431.825,174.488,22.254,153.756
C07105=1081.483,123.123,431.806,174.491,22.257,153.756
C07106=1081.489,123.372,431.786,174.492,22.259,153.756
C07107=1081.494,123.621,431.766,174.494,22.261,153.756
C07108=1081.500,123.871,431.747,174.496,22.263,153.756
C07109=1081.506,124.120,431.727,174.498,22.265,153.756
C07110=1081.512,124.369,431.708,174.500,22.267,153.756
C07111=1081.517,124.618,431.689,174.502,22.269,153.757
C07112=1081.522,124.867,431.669,174.504,22.271,153.757
C07113=1081.528,125.116,431.649,174.505,22.273,153.757
C07114=1081.534,125.365,431.629,174.508,22.275,153.757
C07115=1081.539,125.615,431.610,174.509,22.277,153.757
C07116=1081.545,125.864,431.591,174.511,22.280,153.757
C07117=1081.551,126.113,431.571,174.513,22.282,153.758
C07118=1081.557,126.362,431.552,174.515,22.284,153.758
C07119=1081.563,126.611,431.532,174.517,22.286,153.758
C07120=1081.568,126.861,431.512,174.519,22.288,153.758
C07121=1081.574,127.141,431.490,174.521,22.290,153.758
C07122=1081.581,127.421,431.468,174.523,22.293,153.758
C07123=1081.587,127.700,431.446,174.526,22.295,153.758
C07124=1081.593,127.980,431.424,174.528,22.297,153.759
C07125=1081.599,128.229,431.404,174.529,22.299,153.759
C07126=1081.604,128.479,431.385,174.532,22.302,153.759
C07127=1081.610,128.727,431.365,174.534,22.304,153.759
C07128=1081.616,128.977,431.346,174.535,22.305,153.759
C07129=1081.621,129.226,431.325,174.538,22.308,153.759
C07130=1081.627,129.475,431.305,174.539,22.310,153.759
C07131=1081.633,129.724,431.286,174.541,22.312,153.759
C07132=1081.639,129.973,431.266,174.544,22.314,153.760
C07133=1081.645,130.223,431.247,174.545,22.316,153.760
C07134=1081.651,130.471,431.227,174.548,22.318,153.760
C07135=1081.656,130.722,431.207,174.550,22.320,153.760
C07136=1081.662,130.971,431.187,174.551,22.322,153.760
C07137=1081.668,131.219,431.167,174.554,22.324,153.760
C07138=1081.674,131.469,431.147,174.555,22.326,153.760
C07139=1081.680,131.718,431.128,174.557,22.328,153.760
C07140=1081.685,131.967,431.107,174.560,22.330,153.761
C07141=1081.691,132.216,431.088,174.561,22.332,153.761
C07142=1081.697,132.465,431.068,174.563,22.335,153.761
C07143=1081.702,132.715,431.048,174.565,22.337,153.761
C07144=1081.708,132.964,431.028,174.567,22.339,153.761
C07145=1081.713,133.213,431.007,174.570,22.341,153.761
C07146=1081.719,133.462,430.988,174.571,22.343,153.761
C07147=1081.725,133.711,430.968,174.573,22.345,153.761
C07148=1081.730,133.960,430.948,174.575,22.347,153.762
C07149=1081.736,134.209,430.928,174.577,22.349,153.762
C07150=1081.741,134.459,430.908,174.579,22.351,153.762
C07151=1081.747,134.707,430.888,174.581,22.353,153.762
C07152=1081.752,134.957,430.867,174.583,22.355,153.762
C07153=1081.758,135.205,430.847,174.585,22.357,153.762
C07154=1081.764,135.455,430.828,174.587,22.359,153.762
C07155=1081.769,135.704,430.808,174.589,22.362,153.763
C07156=1081.775,135.953,430.788,174.591,22.364,153.763
C07157=1081.780,136.202,430.767,174.593,22.366,153.763
C07158=1081.786,136.451,430.747,174.595,22.368,153.763
C07159=1081.791,136.700,430.727,174.597,22.370,153.763
C07160=1081.797,136.949,430.707,174.599,22.372,153.763
C07161=1081.803,137.198,430.687,174.601,22.374,153.763
C07162=1081.809,137.448,430.666,174.603,22.376,153.764
C07163=1081.814,137.697,430.646,174.605,22.378,153.764
C07164=1081.820,137.946,430.626,174.607,22.380,153.764
C07165=1081.825,138.196,430.606,174.609,22.382,153.764
C07166=1081.831,138.444,430.586,174.611,22.384,153.764
C07167=1081.837,138.693,430.566,174.613,22.387,153.764
C07168=1081.843,138.942,430.546,174.615,22.388,153.764
C07169=1081.848,139.191,430.525,174.617,22.390,153.764
C07170=1081.854,139.440,430.505,174.619,22.393,153.764
C07171=1081.860,139.690,430.484,174.621,22.395,153.765
C07172=1081.866,139.939,430.464,174.623,22.397,153.765
C07173=1081.871,140.188,430.444,174.626,22.399,153.765
C07174=1081.877,140.437,430.424,174.627,22.401,153.765
C07175=1081.882,140.686,430.403,174.629,22.403,153.765
C07176=1081.887,140.935,430.383,174.632,22.405,153.765
C07177=1081.893,141.184,430.363,174.633,22.407,153.765
C07178=1081.899,141.433,430.342,174.635,22.409,153.765
C07179=1081.904,141.682,430.322,174.638,22.411,153.766
C07180=1081.911,141.932,430.301,174.639,22.413,153.766
C07181=1081.916,142.181,430.281,174.641,22.415,153.766
C07182=1081.921,142.430,430.260,174.644,22.417,153.766
C07183=1081.927,142.679,430.240,174.645,22.419,153.766
C07184=1081.932,142.928,430.220,174.648,22.421,153.766
C07185=1081.939,143.208,430.196,174.650,22.424,153.766
C07186=1081.945,143.488,430.174,174.652,22.426,153.766
C07187=1081.951,143.767,430.151,174.654,22.428,153.767
C07188=1081.957,144.048,430.127,174.657,22.431,153.767
C07189=1081.963,144.297,430.107,174.659,22.433,153.767
C07190=1081.969,144.546,430.087,174.661,22.434,153.767
C07191=1081.974,144.795,430.066,174.663,22.437,153.767
C07192=1081.980,145.045,430.045,174.665,22.439,153.767
C07193=1081.986,145.293,430.025,174.667,22.441,153.767
C07194=1081.991,145.542,430.004,174.669,22.443,153.767
C07195=1081.997,145.791,429.984,174.671,22.445,153.768
C07196=1082.003,146.040,429.964,174.674,22.447,153.768
C07197=1082.008,146.290,429.943,174.675,22.449,153.768
C07198=1082.014,146.539,429.922,174.678,22.451,153.768
C07199=1082.019,146.787,429.901,174.680,22.453,153.768
C07200=1082.025,147.036,429.881,174.681,22.455,153.768
C07201=1082.031,147.286,429.860,174.684,22.457,153.768
C07202=1082.036,147.535,429.839,174.686,22.459,153.768
C07203=1082.042,147.784,429.818,174.688,22.462,153.768
C07204=1082.048,148.032,429.798,174.690,22.463,153.769
C07205=1082.054,148.282,429.777,174.692,22.465,153.769
C07206=1082.059,148.531,429.757,174.694,22.468,153.769
C07207=1082.065,148.780,429.735,174.696,22.469,153.769
C07208=1082.070,149.029,429.715,174.698,22.471,153.769
C07209=1082.076,149.279,429.694,174.701,22.474,153.769
C07210=1082.081,149.527,429.673,174.703,22.476,153.769
C07211=1082.087,149.776,429.653,174.705,22.477,153.769
C07212=1082.093,150.025,429.632,174.707,22.480,153.769
C07213=1082.099,150.274,429.611,174.709,22.482,153.770
C07214=1082.104,150.524,429.590,174.711,22.483,153.770
C07215=1082.109,150.773,429.569,174.713,22.485,153.770
C07216=1082.115,151.021,429.548,174.715,22.488,153.770
C07217=1082.121,151.271,429.527,174.718,22.490,153.770
C07218=1082.126,151.520,429.507,174.719,22.491,153.770
C07219=1082.131,151.769,429.485,174.721,22.494,153.770
C07220=1082.137,152.018,429.465,174.724,22.496,153.770
C07221=1082.143,152.267,429.443,174.725,22.497,153.770
C07222=1082.148,152.516,429.423,174.728,22.500,153.771
C07223=1082.153,152.765,429.402,174.730,22.502,153.771
C07224=1082.160,153.014,429.380,174.732,22.504,153.771
C07225=1082.165,153.264,429.360,174.734,22.506,153.771
C07226=1082.170,153.512,429.339,174.736,22.508,153.771
C07227=1082.176,153.762,429.318,174.739,22.510,153.771
C07228=1082.182,154.010,429.296,174.741,22.512,153.771
C07229=1082.187,154.260,429.276,174.742,22.514,153.771
C07230=1082.193,154.509,429.254,174.745,22.516,153.771
C07231=1082.198,154.758,429.234,174.747,22.518,153.772
C07232=1082.204,155.006,429.212,174.749,22.520,153.772
C07233=1082.210,155.256,429.192,174.751,22.522,153.772
C07234=1082.215,155.505,429.170,174.753,22.524,153.772
C07235=1082.221,155.753,429.149,174.756,22.526,153.772
C07236=1082.227,156.003,429.128,174.758,22.528,153.772
C07237=1082.232,156.252,429.107,174.759,22.530,153.772
C07238=1082.238,156.501,429.086,174.762,22.532,153.772
C07239=1082.244,156.750,429.065,174.764,22.534,153.772
C07240=1082.249,156.999,429.044,174.766,22.536,153.772
C07241=1082.255,157.248,429.022,174.768,22.538,153.773
C07242=1082.261,157.497,429.001,174.770,22.540,153.773
C07243=1082.265,157.746,428.980,174.773,22.542,153.773
C07244=1082.271,157.995,428.958,174.775,22.544,153.773
C07245=1082.277,158.244,428.937,174.777,22.547,153.773
C07246=1082.283,158.494,428.916,174.779,22.548,153.773
C07247=1082.288,158.742,428.895,174.781,22.550,153.773
C07248=1082.294,158.991,428.874,174.784,22.553,153.773
C07249=1082.300,159.271,428.850,174.786,22.555,153.773
C07250=1082.306,159.550,428.826,174.788,22.557,153.773
C07251=1082.313,159.830,428.802,174.791,22.559,153.774
C07252=1082.319,160.110,428.778,174.793,22.561,153.774
C07253=1082.325,160.359,428.756,174.795,22.563,153.774
C07254=1082.330,160.607,428.735,174.798,22.565,153.774
C07255=1082.336,160.857,428.714,174.800,22.568,153.774
C07256=1082.342,161.105,428.693,174.802,22.569,153.774
C07257=1082.348,161.355,428.671,174.804,22.571,153.774
C07258=1082.353,161.603,428.649,174.806,22.573,153.774
C07259=1082.359,161.853,428.628,174.809,22.575,153.774
C07260=1082.363,162.102,428.607,174.811,22.578,153.774
C07261=1082.369,162.351,428.585,174.812,22.580,153.775
C07262=1082.375,162.600,428.564,174.815,22.581,153.775
C07263=1082.380,162.849,428.542,174.817,22.584,153.775
C07264=1082.386,163.098,428.520,174.820,22.586,153.775
C07265=1082.391,163.347,428.499,174.822,22.588,153.775
C07266=1082.396,163.596,428.478,174.823,22.590,153.775
C07267=1082.402,163.845,428.456,174.826,22.592,153.775
C07268=1082.407,164.094,428.434,174.828,22.594,153.775
C07269=1082.413,164.343,428.412,174.831,22.596,153.775
C07270=1082.418,164.592,428.391,174.833,22.598,153.776
C07271=1082.423,164.841,428.369,174.834,22.600,153.776
C07272=1082.429,165.090,428.347,174.837,22.602,153.776
C07273=1082.435,165.338,428.326,174.839,22.604,153.776
C07274=1082.440,165.588,428.304,174.841,22.607,153.776
C07275=1082.446,165.836,428.283,174.844,22.608,153.776
C07276=1082.451,166.086,428.260,174.846,22.611,153.776
C07277=1082.457,166.334,428.239,174.848,22.613,153.776
C07278=1082.462,166.584,428.217,174.850,22.614,153.776
C07279=1082.468,166.832,428.196,174.852,22.617,153.777
C07280=1082.473,167.082,428.173,174.855,22.618,153.777
C07281=1082.479,167.330,428.152,174.857,22.621,153.777
C07282=1082.484,167.580,428.130,174.859,22.623,153.777
C07283=1082.490,167.828,428.109,174.861,22.624,153.777
C07284=1082.495,168.078,428.086,174.863,22.627,153.777
C07285=1082.500,168.327,428.064,174.866,22.629,153.777
C07286=1082.506,168.576,428.043,174.868,22.631,153.777
C07287=1082.511,168.825,428.021,174.870,22.633,153.777
C07288=1082.517,169.074,427.999,174.873,22.635,153.777
